LIN {X 0,Y 544.643,Z 479.184,A -85,B 0,C 180,E1 -3687.041,E2 -3687.041} C_VEL
LIN {X 0,Y 544.543,Z 480.909,A -85,B 0,C 180,E1 -3688.521,E2 -3688.521} C_VEL
LIN {X 0,Y 544.538,Z 481.5,A -85,B 0,C 180,E1 -3690,E2 -3690} C_VEL
LIN {X 0,Y 544.543,Z 480.907,A -85,B 0,C 180,E1 -3691.479,E2 -3691.479} C_VEL
LIN {X 0,Y 544.643,Z 479.179,A -85,B 0,C 180,E1 -3692.959,E2 -3692.959} C_VEL
LIN {X 0,Y 544.606,Z 476.288,A -85,B 0,C 180,E1 -3694.441,E2 -3694.441} C_VEL
LIN {X 0,Y 544.709,Z 472.165,A -85,B 0,C 180,E1 -3695.925,E2 -3695.925} C_VEL
LIN {X 0,Y 544.745,Z 466.7,A -85,B 0,C 180,E1 -3697.413,E2 -3697.413} C_VEL
LIN {X 0,Y 544.845,Z 459.743,A -85,B 0,C 180,E1 -3698.905,E2 -3698.905} C_VEL
LIN {X 0,Y 545.073,Z 451.08,A -85,B 0,C 180,E1 -3700.4,E2 -3700.4} C_VEL
LIN {X 0,Y 545.236,Z 441.69,A -85,B 0,C 180,E1 -3701.734,E2 -3701.734} C_VEL
LIN {X 0,Y 545.476,Z 432.34,A -85,B 0,C 180,E1 -3702.841,E2 -3702.841} C_VEL
LIN {X 0,Y 545.75,Z 421.005,A -85,B 0,C 180,E1 -3703.973,E2 -3703.973} C_VEL
LIN {X 0,Y 546.094,Z 408.349,A -85,B 0,C 180,E1 -3705.028,E2 -3705.028} C_VEL
LIN {X 0,Y 546.426,Z 394.866,A -85,B 0,C 180,E1 -3705.957,E2 -3705.957} C_VEL
LIN {X 0,Y 546.784,Z 381.388,A -85,B 0,C 180,E1 -3706.714,E2 -3706.714} C_VEL
LIN {X 0,Y 547.112,Z 366.588,A -85,B 0,C 180,E1 -3707.377,E2 -3707.377} C_VEL
LIN {X 0,Y 547.36,Z 351.136,A -85,B 0,C 180,E1 -3707.9,E2 -3707.9} C_VEL
LIN {X 0,Y 547.585,Z 335.478,A -85,B 0,C 180,E1 -3708.264,E2 -3708.264} C_VEL
LIN {X 0,Y 547.881,Z 279.91,A -85,B 0,C 180,E1 -3709.045,E2 -3709.045} C_VEL
LIN {X 0,Y 548.382,Z 177.465,A -85,B 0,C 180,E1 -3710.426,E2 -3710.426} C_VEL
LIN {X 0,Y 546.956,Z 166.898,A -85,B 0,C 180,E1 -3710.651,E2 -3710.651} C_VEL
LIN {X 0,Y 547.549,Z 134.253,A -85,B 0,C 180,E1 -3713.647,E2 -3713.647} C_VEL
LIN {X 0,Y 548.011,Z 115.051,A -85,B 0,C 180,E1 -3715.43,E2 -3715.43} C_VEL
LIN {X 0,Y 545.068,Z 103.217,A -85,B 0,C 180,E1 -3716.723,E2 -3716.723} C_VEL
LIN {X 0,Y 545.02,Z 103.223,A -85,B 0,C 180,E1 -3719.341,E2 -3719.341} C_VEL
LIN {X 0,Y 545.044,Z 103.214,A -85,B 0,C 180,E1 -3721.916,E2 -3721.916} C_VEL
LIN {X 0,Y 545.045,Z 103.216,A -85,B 0,C 180,E1 -3724.566,E2 -3724.566} C_VEL
LIN {X 0,Y 545.029,Z 103.22,A -85,B 0,C 180,E1 -3727.305,E2 -3727.305} C_VEL
LIN {X 0,Y 545.061,Z 103.212,A -85,B 0,C 180,E1 -3730.143,E2 -3730.143} C_VEL
LIN {X 0,Y 545.016,Z 103.22,A -85,B 0,C 180,E1 -3733.113,E2 -3733.113} C_VEL
LIN {X 0,Y 545.027,Z 103.216,A -85,B 0,C 180,E1 -3736.229,E2 -3736.229} C_VEL
LIN {X 0,Y 545.027,Z 103.22,A -85,B 0,C 180,E1 -3738.881,E2 -3738.881} C_VEL
LIN {X 0,Y 545.045,Z 103.214,A -85,B 0,C 180,E1 -3741.762,E2 -3741.762} C_VEL
LIN {X 0,Y 545.024,Z 103.223,A -85,B 0,C 180,E1 -3744.531,E2 -3744.531} C_VEL
LIN {X 0,Y 545.061,Z 103.212,A -85,B 0,C 180,E1 -3747.211,E2 -3747.211} C_VEL
LIN {X 0,Y 545.062,Z 103.213,A -85,B 0,C 180,E1 -3749.811,E2 -3749.811} C_VEL
LIN {X 0,Y 545.039,Z 103.217,A -85,B 0,C 180,E1 -3752.838,E2 -3752.838} C_VEL
LIN {X 0,Y 545.021,Z 103.22,A -85,B 0,C 180,E1 -3755.63,E2 -3755.63} C_VEL
LIN {X 0,Y 545.071,Z 103.293,A -85,B 0,C 180,E1 -3757.943,E2 -3757.943} C_VEL
LIN {X 0,Y 546.269,Z 110.508,A -85,B 0,C 180,E1 -3759.063,E2 -3759.063} C_VEL
LIN {X 0,Y 546.308,Z 113.04,A -85,B 0,C 180,E1 -3759.438,E2 -3759.438} C_VEL
LIN {X 0,Y 548.468,Z 123.652,A -85,B 0,C 180,E1 -3759.681,E2 -3759.681} C_VEL
LIN {X 0,Y 547.486,Z 277.991,A -85,B 0,C 180,E1 -3761.845,E2 -3761.845} C_VEL
LIN {X 0,Y 547.341,Z 292.858,A -85,B 0,C 180,E1 -3762.196,E2 -3762.196} C_VEL
LIN {X 0,Y 547.079,Z 308.282,A -85,B 0,C 180,E1 -3762.718,E2 -3762.718} C_VEL
LIN {X 0,Y 546.831,Z 321.071,A -85,B 0,C 180,E1 -3763.288,E2 -3763.288} C_VEL
LIN {X 0,Y 546.499,Z 334.745,A -85,B 0,C 180,E1 -3764.045,E2 -3764.045} C_VEL
LIN {X 0,Y 546.16,Z 348.31,A -85,B 0,C 180,E1 -3764.973,E2 -3764.973} C_VEL
LIN {X 0,Y 545.791,Z 360.976,A -85,B 0,C 180,E1 -3766.029,E2 -3766.029} C_VEL
LIN {X 0,Y 545.513,Z 372.228,A -85,B 0,C 180,E1 -3767.16,E2 -3767.16} C_VEL
LIN {X 0,Y 545.253,Z 382.568,A -85,B 0,C 180,E1 -3768.407,E2 -3768.407} C_VEL
LIN {X 0,Y 545.092,Z 390.911,A -85,B 0,C 180,E1 -3769.601,E2 -3769.601} C_VEL
LIN {X 0,Y 544.851,Z 399.516,A -85,B 0,C 180,E1 -3771.096,E2 -3771.096} C_VEL
LIN {X 0,Y 544.746,Z 406.525,A -85,B 0,C 180,E1 -3772.588,E2 -3772.588} C_VEL
LIN {X 0,Y 544.708,Z 411.986,A -85,B 0,C 180,E1 -3774.076,E2 -3774.076} C_VEL
LIN {X 0,Y 544.605,Z 416.188,A -85,B 0,C 180,E1 -3775.559,E2 -3775.559} C_VEL
LIN {X 0,Y 544.643,Z 419.108,A -85,B 0,C 180,E1 -3777.042,E2 -3777.042} C_VEL
LIN {X 0,Y 544.542,Z 420.838,A -85,B 0,C 180,E1 -3778.521,E2 -3778.521} C_VEL
LIN {X 0,Y 544.539,Z 421.496,A -85,B 0,C 180,E1 -3780,E2 -3780} C_VEL
LIN {X 0,Y 544.544,Z 420.915,A -85,B 0,C 180,E1 -3781.479,E2 -3781.479} C_VEL
LIN {X 0,Y 544.645,Z 419.238,A -85,B 0,C 180,E1 -3782.959,E2 -3782.959} C_VEL
LIN {X 0,Y 544.606,Z 416.423,A -85,B 0,C 180,E1 -3784.441,E2 -3784.441} C_VEL
LIN {X 0,Y 544.701,Z 412.267,A -85,B 0,C 180,E1 -3785.925,E2 -3785.925} C_VEL
LIN {X 0,Y 544.743,Z 406.901,A -85,B 0,C 180,E1 -3787.413,E2 -3787.413} C_VEL
LIN {X 0,Y 544.846,Z 399.966,A -85,B 0,C 180,E1 -3788.905,E2 -3788.905} C_VEL
LIN {X 0,Y 545.047,Z 392.645,A -85,B 0,C 180,E1 -3790.213,E2 -3790.213} C_VEL
LIN {X 0,Y 545.165,Z 383.552,A -85,B 0,C 180,E1 -3791.549,E2 -3791.549} C_VEL
LIN {X 0,Y 545.442,Z 374.644,A -85,B 0,C 180,E1 -3792.653,E2 -3792.653} C_VEL
LIN {X 0,Y 545.757,Z 362.903,A -85,B 0,C 180,E1 -3793.878,E2 -3793.878} C_VEL
LIN {X 0,Y 546.104,Z 350.94,A -85,B 0,C 180,E1 -3794.915,E2 -3794.915} C_VEL
LIN {X 0,Y 546.421,Z 337.749,A -85,B 0,C 180,E1 -3795.862,E2 -3795.862} C_VEL
LIN {X 0,Y 546.759,Z 324.87,A -85,B 0,C 180,E1 -3796.619,E2 -3796.619} C_VEL
LIN {X 0,Y 547.089,Z 310.858,A -85,B 0,C 180,E1 -3797.282,E2 -3797.282} C_VEL
LIN {X 0,Y 547.355,Z 295.027,A -85,B 0,C 180,E1 -3797.852,E2 -3797.852} C_VEL
LIN {X 0,Y 547.539,Z 279.859,A -85,B 0,C 180,E1 -3798.235,E2 -3798.235} C_VEL
LIN {X 0,Y 547.672,Z 258.394,A -85,B 0,C 180,E1 -3798.561,E2 -3798.561} C_VEL
LIN {X 0,Y 548.302,Z 149.592,A -85,B 0,C 180,E1 -3800.048,E2 -3800.048} C_VEL
LIN {X 0,Y 547.879,Z 143.779,A -85,B 0,C 180,E1 -3800.144,E2 -3800.144} C_VEL
LIN {X 0,Y 545.529,Z 134.425,A -85,B 0,C 180,E1 -3800.368,E2 -3800.368} C_VEL
LIN {X 0,Y 540.885,Z 119.579,A -85,B 0,C 180,E1 -3800.769,E2 -3800.769} C_VEL
LIN {X 0,Y 539.323,Z 112.564,A -85,B 0,C 180,E1 -3800.944,E2 -3800.944} C_VEL
LIN {X 0,Y 538.741,Z 107.608,A -85,B 0,C 180,E1 -3801.726,E2 -3801.726} C_VEL
LIN {X 0,Y 538.019,Z 104.095,A -85,B 0,C 180,E1 -3802.311,E2 -3802.311} C_VEL
LIN {X 0,Y 538.03,Z 104.093,A -85,B 0,C 180,E1 -3805.535,E2 -3805.535} C_VEL
LIN {X 0,Y 537.997,Z 104.095,A -85,B 0,C 180,E1 -3808.053,E2 -3808.053} C_VEL
LIN {X 0,Y 538.009,Z 104.089,A -85,B 0,C 180,E1 -3810.628,E2 -3810.628} C_VEL
LIN {X 0,Y 538.022,Z 104.092,A -85,B 0,C 180,E1 -3813.279,E2 -3813.279} C_VEL
LIN {X 0,Y 537.99,Z 104.094,A -85,B 0,C 180,E1 -3816.005,E2 -3816.005} C_VEL
LIN {X 0,Y 538.011,Z 104.089,A -85,B 0,C 180,E1 -3818.831,E2 -3818.831} C_VEL
LIN {X 0,Y 537.991,Z 104.093,A -85,B 0,C 180,E1 -3821.874,E2 -3821.874} C_VEL
LIN {X 0,Y 537.996,Z 104.091,A -85,B 0,C 180,E1 -3824.864,E2 -3824.864} C_VEL
LIN {X 0,Y 537.976,Z 104.093,A -85,B 0,C 180,E1 -3827.21,E2 -3827.21} C_VEL
LIN {X 0,Y 538.01,Z 104.088,A -85,B 0,C 180,E1 -3830.202,E2 -3830.202} C_VEL
LIN {X 0,Y 538.021,Z 104.092,A -85,B 0,C 180,E1 -3833.067,E2 -3833.067} C_VEL
LIN {X 0,Y 538,Z 104.088,A -85,B 0,C 180,E1 -3835.825,E2 -3835.825} C_VEL
LIN {X 0,Y 537.993,Z 104.093,A -85,B 0,C 180,E1 -3838.498,E2 -3838.498} C_VEL
LIN {X 0,Y 537.987,Z 104.096,A -85,B 0,C 180,E1 -3841.096,E2 -3841.096} C_VEL
LIN {X 0,Y 537.992,Z 104.091,A -85,B 0,C 180,E1 -3843.631,E2 -3843.631} C_VEL
LIN {X 0,Y 537.987,Z 104.089,A -85,B 0,C 180,E1 -3846.128,E2 -3846.128} C_VEL
LIN {X 0,Y 538.001,Z 104.097,A -85,B 0,C 180,E1 -3848.545,E2 -3848.545} C_VEL
LIN {X 0,Y 538.009,Z 104.094,A -85,B 0,C 180,E1 -3850.939,E2 -3850.939} C_VEL
LIN {X 0,Y 537.972,Z 104.092,A -85,B 0,C 180,E1 -3853.297,E2 -3853.297} C_VEL
LIN {X 0,Y 538.037,Z 104.086,A -85,B 0,C 180,E1 -3855.63,E2 -3855.63} C_VEL
LIN {X 0,Y 538.079,Z 104.084,A -85,B 0,C 180,E1 -3858.702,E2 -3858.702} C_VEL
LIN {X 0,Y 538.037,Z 104.087,A -85,B 0,C 180,E1 -3861.739,E2 -3861.739} C_VEL
LIN {X 0,Y 538.122,Z 104.079,A -85,B 0,C 180,E1 -3864.755,E2 -3864.755} C_VEL
LIN {X 0,Y 538.163,Z 104.075,A -85,B 0,C 180,E1 -3867.755,E2 -3867.755} C_VEL
LIN {X 0,Y 538.162,Z 104.078,A -85,B 0,C 180,E1 -3870,E2 -3870} C_VEL
LIN {X 0,Y 538.021,Z 104.191,A -85,B 0,C 180,E1 -3871.193,E2 -3871.193} C_VEL
LIN {X 0,Y 539.86,Z 112.82,A -85,B 0,C 180,E1 -3872.425,E2 -3872.425} C_VEL
LIN {X 0,Y 539.768,Z 126.914,A -85,B 0,C 180,E1 -3874.294,E2 -3874.294} C_VEL
LIN {X 0,Y 539.542,Z 141.011,A -85,B 0,C 180,E1 -3876.146,E2 -3876.146} C_VEL
LIN {X 0,Y 541.815,Z 152.663,A -85,B 0,C 180,E1 -3876.4,E2 -3876.4} C_VEL
LIN {X 0,Y 540.966,Z 306.907,A -85,B 0,C 180,E1 -3878.521,E2 -3878.521} C_VEL
LIN {X 0,Y 540.76,Z 321.623,A -85,B 0,C 180,E1 -3878.871,E2 -3878.871} C_VEL
LIN {X 0,Y 540.477,Z 336.09,A -85,B 0,C 180,E1 -3879.354,E2 -3879.354} C_VEL
LIN {X 0,Y 540.088,Z 351.048,A -85,B 0,C 180,E1 -3880.023,E2 -3880.023} C_VEL
LIN {X 0,Y 539.762,Z 362.973,A -85,B 0,C 180,E1 -3880.693,E2 -3880.693} C_VEL
LIN {X 0,Y 539.431,Z 374.357,A -85,B 0,C 180,E1 -3881.458,E2 -3881.458} C_VEL
LIN {X 0,Y 539.062,Z 385.999,A -85,B 0,C 180,E1 -3882.384,E2 -3882.384} C_VEL
LIN {X 0,Y 538.682,Z 398.586,A -85,B 0,C 180,E1 -3883.582,E2 -3883.582} C_VEL
LIN {X 0,Y 538.352,Z 407.929,A -85,B 0,C 180,E1 -3884.649,E2 -3884.649} C_VEL
LIN {X 0,Y 538.123,Z 416.015,A -85,B 0,C 180,E1 -3885.724,E2 -3885.724} C_VEL
LIN {X 0,Y 537.955,Z 423.592,A -85,B 0,C 180,E1 -3886.895,E2 -3886.895} C_VEL
LIN {X 0,Y 537.811,Z 430.113,A -85,B 0,C 180,E1 -3888.081,E2 -3888.081} C_VEL
LIN {X 0,Y 537.672,Z 436.272,A -85,B 0,C 180,E1 -3889.415,E2 -3889.415} C_VEL
LIN {X 0,Y 537.576,Z 442.31,A -85,B 0,C 180,E1 -3891.071,E2 -3891.071} C_VEL
LIN {X 0,Y 537.519,Z 445.693,A -85,B 0,C 180,E1 -3892.282,E2 -3892.282} C_VEL
LIN {X 0,Y 537.44,Z 448.666,A -85,B 0,C 180,E1 -3893.74,E2 -3893.74} C_VEL
LIN {X 0,Y 537.421,Z 450.12,A -85,B 0,C 180,E1 -3894.738,E2 -3894.738} C_VEL
LIN {X 0,Y 537.457,Z 450.902,A -85,B 0,C 180,E1 -3895.564,E2 -3895.564} C_VEL
LIN {X 0,Y 537.457,Z 451.454,A -85,B 0,C 180,E1 -3897.237,E2 -3897.237} C_VEL
LIN {X 0,Y 537.474,Z 450.617,A -85,B 0,C 180,E1 -3898.825,E2 -3898.825} C_VEL
LIN {X 0,Y 537.514,Z 448.664,A -85,B 0,C 180,E1 -3900.35,E2 -3900.35} C_VEL
LIN {X 0,Y 537.539,Z 445.699,A -85,B 0,C 180,E1 -3901.805,E2 -3901.805} C_VEL
LIN {X 0,Y 537.583,Z 441.423,A -85,B 0,C 180,E1 -3903.304,E2 -3903.304} C_VEL
LIN {X 0,Y 537.678,Z 435.709,A -85,B 0,C 180,E1 -3904.806,E2 -3904.806} C_VEL
LIN {X 0,Y 537.777,Z 430.06,A -85,B 0,C 180,E1 -3906.021,E2 -3906.021} C_VEL
LIN {X 0,Y 537.919,Z 423.829,A -85,B 0,C 180,E1 -3907.157,E2 -3907.157} C_VEL
LIN {X 0,Y 538.103,Z 417.58,A -85,B 0,C 180,E1 -3908.14,E2 -3908.14} C_VEL
LIN {X 0,Y 538.285,Z 409.15,A -85,B 0,C 180,E1 -3909.289,E2 -3909.289} C_VEL
LIN {X 0,Y 538.641,Z 398.911,A -85,B 0,C 180,E1 -3910.475,E2 -3910.475} C_VEL
LIN {X 0,Y 539.034,Z 386.361,A -85,B 0,C 180,E1 -3911.678,E2 -3911.678} C_VEL
LIN {X 0,Y 539.395,Z 375.415,A -85,B 0,C 180,E1 -3912.557,E2 -3912.557} C_VEL
LIN {X 0,Y 539.719,Z 364.092,A -85,B 0,C 180,E1 -3913.329,E2 -3913.329} C_VEL
LIN {X 0,Y 540.113,Z 350.528,A -85,B 0,C 180,E1 -3914.095,E2 -3914.095} C_VEL
LIN {X 0,Y 540.468,Z 336.169,A -85,B 0,C 180,E1 -3914.734,E2 -3914.734} C_VEL
LIN {X 0,Y 540.751,Z 321.821,A -85,B 0,C 180,E1 -3915.214,E2 -3915.214} C_VEL
LIN {X 0,Y 540.97,Z 308.257,A -85,B 0,C 180,E1 -3915.542,E2 -3915.542} C_VEL
LIN {X 0,Y 541.146,Z 275.268,A -85,B 0,C 180,E1 -3916.019,E2 -3916.019} C_VEL
LIN {X 0,Y 541.751,Z 148.68,A -85,B 0,C 180,E1 -3917.748,E2 -3917.748} C_VEL
LIN {X 0,Y 540.144,Z 139.429,A -85,B 0,C 180,E1 -3917.959,E2 -3917.959} C_VEL
LIN {X 0,Y 540.434,Z 114.155,A -85,B 0,C 180,E1 -3920.536,E2 -3920.536} C_VEL
LIN {X 0,Y 538.019,Z 104.094,A -85,B 0,C 180,E1 -3921.693,E2 -3921.693} C_VEL
LIN {X 0,Y 537.992,Z 104.098,A -85,B 0,C 180,E1 -3924.089,E2 -3924.089} C_VEL
LIN {X 0,Y 538.033,Z 104.088,A -85,B 0,C 180,E1 -3926.727,E2 -3926.727} C_VEL
LIN {X 0,Y 538.029,Z 104.093,A -85,B 0,C 180,E1 -3929.556,E2 -3929.556} C_VEL
LIN {X 0,Y 538.043,Z 104.09,A -85,B 0,C 180,E1 -3931.95,E2 -3931.95} C_VEL
LIN {X 0,Y 538.074,Z 104.083,A -85,B 0,C 180,E1 -3934.467,E2 -3934.467} C_VEL
LIN {X 0,Y 537.996,Z 104.099,A -85,B 0,C 180,E1 -3937.738,E2 -3937.738} C_VEL
LIN {X 0,Y 538.046,Z 104.233,A -85,B 0,C 180,E1 -3938.194,E2 -3938.194} C_VEL
LIN {X 0,Y 539.646,Z 111.177,A -85,B 0,C 180,E1 -3939.135,E2 -3939.135} C_VEL
LIN {X 0,Y 541.692,Z 120.025,A -85,B 0,C 180,E1 -3939.352,E2 -3939.352} C_VEL
LIN {X 0,Y 541.213,Z 211.695,A -85,B 0,C 180,E1 -3940.662,E2 -3940.662} C_VEL
LIN {X 0,Y 540.755,Z 277.646,A -85,B 0,C 180,E1 -3941.593,E2 -3941.593} C_VEL
LIN {X 0,Y 540.575,Z 293.955,A -85,B 0,C 180,E1 -3941.99,E2 -3941.99} C_VEL
LIN {X 0,Y 540.278,Z 308.349,A -85,B 0,C 180,E1 -3942.493,E2 -3942.493} C_VEL
LIN {X 0,Y 540.006,Z 321.097,A -85,B 0,C 180,E1 -3943.07,E2 -3943.07} C_VEL
LIN {X 0,Y 539.638,Z 334.778,A -85,B 0,C 180,E1 -3943.836,E2 -3943.836} C_VEL
LIN {X 0,Y 539.285,Z 348.853,A -85,B 0,C 180,E1 -3944.815,E2 -3944.815} C_VEL
LIN {X 0,Y 538.903,Z 359.967,A -85,B 0,C 180,E1 -3945.75,E2 -3945.75} C_VEL
LIN {X 0,Y 538.607,Z 370.522,A -85,B 0,C 180,E1 -3946.8,E2 -3946.8} C_VEL
LIN {X 0,Y 538.31,Z 380.347,A -85,B 0,C 180,E1 -3947.942,E2 -3947.942} C_VEL
LIN {X 0,Y 538.072,Z 391.099,A -85,B 0,C 180,E1 -3949.463,E2 -3949.463} C_VEL
LIN {X 0,Y 537.856,Z 397.775,A -85,B 0,C 180,E1 -3950.599,E2 -3950.599} C_VEL
LIN {X 0,Y 537.768,Z 403.459,A -85,B 0,C 180,E1 -3951.734,E2 -3951.734} C_VEL
LIN {X 0,Y 537.679,Z 408.25,A -85,B 0,C 180,E1 -3952.867,E2 -3952.867} C_VEL
LIN {X 0,Y 537.643,Z 413.347,A -85,B 0,C 180,E1 -3954.373,E2 -3954.373} C_VEL
LIN {X 0,Y 537.562,Z 418,A -85,B 0,C 180,E1 -3956.252,E2 -3956.252} C_VEL
LIN {X 0,Y 537.488,Z 420.262,A -85,B 0,C 180,E1 -3957.752,E2 -3957.752} C_VEL
LIN {X 0,Y 537.439,Z 421.392,A -85,B 0,C 180,E1 -3959.25,E2 -3959.25} C_VEL
LIN {X 0,Y 537.441,Z 421.625,A -85,B 0,C 180,E1 -3960,E2 -3960} C_VEL
LIN {X 0,Y 537.449,Z 421.076,A -85,B 0,C 180,E1 -3961.498,E2 -3961.498} C_VEL
LIN {X 0,Y 537.574,Z 419.381,A -85,B 0,C 180,E1 -3962.997,E2 -3962.997} C_VEL
LIN {X 0,Y 537.562,Z 418.182,A -85,B 0,C 180,E1 -3963.748,E2 -3963.748} C_VEL
LIN {X 0,Y 537.643,Z 413.645,A -85,B 0,C 180,E1 -3965.626,E2 -3965.626} C_VEL
LIN {X 0,Y 537.68,Z 408.627,A -85,B 0,C 180,E1 -3967.133,E2 -3967.133} C_VEL
LIN {X 0,Y 537.778,Z 402.213,A -85,B 0,C 180,E1 -3968.643,E2 -3968.643} C_VEL
LIN {X 0,Y 537.984,Z 394.053,A -85,B 0,C 180,E1 -3970.157,E2 -3970.157} C_VEL
LIN {X 0,Y 538.09,Z 386.69,A -85,B 0,C 180,E1 -3971.298,E2 -3971.298} C_VEL
LIN {X 0,Y 538.374,Z 378.069,A -85,B 0,C 180,E1 -3972.438,E2 -3972.438} C_VEL
LIN {X 0,Y 538.7,Z 367.876,A -85,B 0,C 180,E1 -3973.582,E2 -3973.582} C_VEL
LIN {X 0,Y 539.029,Z 355.64,A -85,B 0,C 180,E1 -3974.729,E2 -3974.729} C_VEL
LIN {X 0,Y 539.411,Z 343.304,A -85,B 0,C 180,E1 -3975.683,E2 -3975.683} C_VEL
LIN {X 0,Y 539.757,Z 329.755,A -85,B 0,C 180,E1 -3976.548,E2 -3976.548} C_VEL
LIN {X 0,Y 540.09,Z 315.713,A -85,B 0,C 180,E1 -3977.268,E2 -3977.268} C_VEL
LIN {X 0,Y 540.388,Z 300.471,A -85,B 0,C 180,E1 -3977.869,E2 -3977.869} C_VEL
LIN {X 0,Y 540.641,Z 284.928,A -85,B 0,C 180,E1 -3978.312,E2 -3978.312} C_VEL
LIN {X 0,Y 540.764,Z 268.903,A -85,B 0,C 180,E1 -3978.602,E2 -3978.602} C_VEL
LIN {X 0,Y 541.688,Z 140.378,A -85,B 0,C 180,E1 -3980.429,E2 -3980.429} C_VEL
LIN {X 0,Y 541.716,Z 123.174,A -85,B 0,C 180,E1 -3980.691,E2 -3980.691} C_VEL
LIN {X 0,Y 539.622,Z 114.321,A -85,B 0,C 180,E1 -3980.928,E2 -3980.928} C_VEL
LIN {X 0,Y 539.443,Z 110.534,A -85,B 0,C 180,E1 -3981.567,E2 -3981.567} C_VEL
LIN {X 0,Y 537.987,Z 104.098,A -85,B 0,C 180,E1 -3982.768,E2 -3982.768} C_VEL
LIN {X 0,Y 538.007,Z 104.097,A -85,B 0,C 180,E1 -3985.664,E2 -3985.664} C_VEL
LIN {X 0,Y 537.996,Z 104.097,A -85,B 0,C 180,E1 -3988.052,E2 -3988.052} C_VEL
LIN {X 0,Y 538.007,Z 104.091,A -85,B 0,C 180,E1 -3990.628,E2 -3990.628} C_VEL
LIN {X 0,Y 538.019,Z 104.094,A -85,B 0,C 180,E1 -3993.278,E2 -3993.278} C_VEL
LIN {X 0,Y 537.987,Z 104.095,A -85,B 0,C 180,E1 -3996.005,E2 -3996.005} C_VEL
LIN {X 0,Y 538.008,Z 104.092,A -85,B 0,C 180,E1 -3998.831,E2 -3998.831} C_VEL
LIN {X 0,Y 537.987,Z 104.095,A -85,B 0,C 180,E1 -4001.873,E2 -4001.873} C_VEL
LIN {X 0,Y 537.993,Z 104.096,A -85,B 0,C 180,E1 -4004.863,E2 -4004.863} C_VEL
LIN {X 0,Y 537.973,Z 104.101,A -85,B 0,C 180,E1 -4007.209,E2 -4007.209} C_VEL
LIN {X 0,Y 538.006,Z 104.091,A -85,B 0,C 180,E1 -4010.201,E2 -4010.201} C_VEL
LIN {X 0,Y 538.016,Z 104.097,A -85,B 0,C 180,E1 -4013.066,E2 -4013.066} C_VEL
LIN {X 0,Y 537.995,Z 104.093,A -85,B 0,C 180,E1 -4015.825,E2 -4015.825} C_VEL
LIN {X 0,Y 537.988,Z 104.099,A -85,B 0,C 180,E1 -4018.497,E2 -4018.497} C_VEL
LIN {X 0,Y 537.984,Z 104.119,A -85,B 0,C 180,E1 -4021.415,E2 -4021.415} C_VEL
LIN {X 0,Y 540.297,Z 114.01,A -85,B 0,C 180,E1 -4022.774,E2 -4022.774} C_VEL
LIN {X 0,Y 540.209,Z 127.243,A -85,B 0,C 180,E1 -4024.389,E2 -4024.389} C_VEL
LIN {X 0,Y 539.701,Z 152.43,A -85,B 0,C 180,E1 -4027.372,E2 -4027.372} C_VEL
LIN {X 0,Y 539.403,Z 167.004,A -85,B 0,C 180,E1 -4029.066,E2 -4029.066} C_VEL
LIN {X 0,Y 541.666,Z 181.231,A -85,B 0,C 180,E1 -4029.388,E2 -4029.388} C_VEL
LIN {X 0,Y 540.901,Z 297.15,A -85,B 0,C 180,E1 -4031.02,E2 -4031.02} C_VEL
LIN {X 0,Y 540.627,Z 336.129,A -85,B 0,C 180,E1 -4031.586,E2 -4031.586} C_VEL
LIN {X 0,Y 540.429,Z 351.514,A -85,B 0,C 180,E1 -4031.961,E2 -4031.961} C_VEL
LIN {X 0,Y 540.147,Z 365.617,A -85,B 0,C 180,E1 -4032.44,E2 -4032.44} C_VEL
LIN {X 0,Y 539.837,Z 379.671,A -85,B 0,C 180,E1 -4033.065,E2 -4033.065} C_VEL
LIN {X 0,Y 539.411,Z 393.424,A -85,B 0,C 180,E1 -4033.83,E2 -4033.83} C_VEL
LIN {X 0,Y 539.106,Z 407.383,A -85,B 0,C 180,E1 -4034.787,E2 -4034.787} C_VEL
LIN {X 0,Y 538.733,Z 420.06,A -85,B 0,C 180,E1 -4035.842,E2 -4035.842} C_VEL
LIN {X 0,Y 538.433,Z 431.551,A -85,B 0,C 180,E1 -4036.988,E2 -4036.988} C_VEL
LIN {X 0,Y 538.148,Z 442.074,A -85,B 0,C 180,E1 -4038.241,E2 -4038.241} C_VEL
LIN {X 0,Y 537.985,Z 451.91,A -85,B 0,C 180,E1 -4039.652,E2 -4039.652} C_VEL
LIN {X 0,Y 537.797,Z 459.537,A -85,B 0,C 180,E1 -4040.978,E2 -4040.978} C_VEL
LIN {X 0,Y 537.661,Z 466.643,A -85,B 0,C 180,E1 -4042.489,E2 -4042.489} C_VEL
LIN {X 0,Y 537.623,Z 472.161,A -85,B 0,C 180,E1 -4043.997,E2 -4043.997} C_VEL
LIN {X 0,Y 537.508,Z 476.29,A -85,B 0,C 180,E1 -4045.5,E2 -4045.5} C_VEL
LIN {X 0,Y 537.543,Z 479.183,A -85,B 0,C 180,E1 -4047.002,E2 -4047.002} C_VEL
LIN {X 0,Y 537.448,Z 480.909,A -85,B 0,C 180,E1 -4048.501,E2 -4048.501} C_VEL
LIN {X 0,Y 537.439,Z 481.5,A -85,B 0,C 180,E1 -4050,E2 -4050} C_VEL
LIN {X 0,Y 537.448,Z 480.906,A -85,B 0,C 180,E1 -4051.499,E2 -4051.499} C_VEL
LIN {X 0,Y 537.543,Z 479.178,A -85,B 0,C 180,E1 -4052.998,E2 -4052.998} C_VEL
LIN {X 0,Y 537.508,Z 476.287,A -85,B 0,C 180,E1 -4054.5,E2 -4054.5} C_VEL
LIN {X 0,Y 537.623,Z 472.165,A -85,B 0,C 180,E1 -4056.003,E2 -4056.003} C_VEL
LIN {X 0,Y 537.661,Z 466.645,A -85,B 0,C 180,E1 -4057.511,E2 -4057.511} C_VEL
LIN {X 0,Y 537.797,Z 459.558,A -85,B 0,C 180,E1 -4059.022,E2 -4059.022} C_VEL
LIN {X 0,Y 538.005,Z 450.726,A -85,B 0,C 180,E1 -4060.538,E2 -4060.538} C_VEL
LIN {X 0,Y 538.204,Z 440.976,A -85,B 0,C 180,E1 -4061.912,E2 -4061.912} C_VEL
LIN {X 0,Y 538.443,Z 431.755,A -85,B 0,C 180,E1 -4063.012,E2 -4063.012} C_VEL
LIN {X 0,Y 538.75,Z 420.377,A -85,B 0,C 180,E1 -4064.158,E2 -4064.158} C_VEL
LIN {X 0,Y 539.138,Z 407.558,A -85,B 0,C 180,E1 -4065.234,E2 -4065.234} C_VEL
LIN {X 0,Y 539.487,Z 394.091,A -85,B 0,C 180,E1 -4066.168,E2 -4066.168} C_VEL
LIN {X 0,Y 539.877,Z 380.546,A -85,B 0,C 180,E1 -4066.934,E2 -4066.934} C_VEL
LIN {X 0,Y 540.246,Z 365.604,A -85,B 0,C 180,E1 -4067.605,E2 -4067.605} C_VEL
LIN {X 0,Y 540.543,Z 349.885,A -85,B 0,C 180,E1 -4068.133,E2 -4068.133} C_VEL
LIN {X 0,Y 540.789,Z 334.296,A -85,B 0,C 180,E1 -4068.492,E2 -4068.492} C_VEL
LIN {X 0,Y 541.185,Z 271.432,A -85,B 0,C 180,E1 -4069.388,E2 -4069.388} C_VEL
LIN {X 0,Y 541.704,Z 178.455,A -85,B 0,C 180,E1 -4070.669,E2 -4070.669} C_VEL
LIN {X 0,Y 540.108,Z 166.532,A -85,B 0,C 180,E1 -4070.93,E2 -4070.93} C_VEL
LIN {X 0,Y 540.802,Z 134.049,A -85,B 0,C 180,E1 -4073.952,E2 -4073.952} C_VEL
LIN {X 0,Y 541.258,Z 117.243,A -85,B 0,C 180,E1 -4075.531,E2 -4075.531} C_VEL
LIN {X 0,Y 539.353,Z 109.176,A -85,B 0,C 180,E1 -4076.402,E2 -4076.402} C_VEL
LIN {X 0,Y 538.011,Z 104.097,A -85,B 0,C 180,E1 -4076.97,E2 -4076.97} C_VEL
LIN {X 0,Y 537.996,Z 104.094,A -85,B 0,C 180,E1 -4079.762,E2 -4079.762} C_VEL
LIN {X 0,Y 538.01,Z 104.091,A -85,B 0,C 180,E1 -4082.383,E2 -4082.383} C_VEL
LIN {X 0,Y 537.985,Z 104.099,A -85,B 0,C 180,E1 -4085.085,E2 -4085.085} C_VEL
LIN {X 0,Y 537.986,Z 104.093,A -85,B 0,C 180,E1 -4087.878,E2 -4087.878} C_VEL
LIN {X 0,Y 538.001,Z 104.097,A -85,B 0,C 180,E1 -4090.78,E2 -4090.78} C_VEL
LIN {X 0,Y 538,Z 104.09,A -85,B 0,C 180,E1 -4094.071,E2 -4094.071} C_VEL
LIN {X 0,Y 537.97,Z 104.098,A -85,B 0,C 180,E1 -4097.019,E2 -4097.019} C_VEL
LIN {X 0,Y 538.005,Z 104.091,A -85,B 0,C 180,E1 -4099.258,E2 -4099.258} C_VEL
LIN {X 0,Y 537.986,Z 104.096,A -85,B 0,C 180,E1 -4102.122,E2 -4102.122} C_VEL
LIN {X 0,Y 537.986,Z 104.096,A -85,B 0,C 180,E1 -4104.915,E2 -4104.915} C_VEL
LIN {X 0,Y 538.014,Z 104.09,A -85,B 0,C 180,E1 -4107.617,E2 -4107.617} C_VEL
LIN {X 0,Y 537.999,Z 104.098,A -85,B 0,C 180,E1 -4110.238,E2 -4110.238} C_VEL
LIN {X 0,Y 538.012,Z 104.094,A -85,B 0,C 180,E1 -4112.793,E2 -4112.793} C_VEL
LIN {X 0,Y 537.983,Z 104.096,A -85,B 0,C 180,E1 -4115.29,E2 -4115.29} C_VEL
LIN {X 0,Y 538.049,Z 104.182,A -85,B 0,C 180,E1 -4117.741,E2 -4117.741} C_VEL
LIN {X 0,Y 539.422,Z 111.104,A -85,B 0,C 180,E1 -4118.805,E2 -4118.805} C_VEL
LIN {X 0,Y 539.539,Z 113.837,A -85,B 0,C 180,E1 -4119.183,E2 -4119.183} C_VEL
LIN {X 0,Y 541.81,Z 124.5,A -85,B 0,C 180,E1 -4119.436,E2 -4119.436} C_VEL
LIN {X 0,Y 540.676,Z 277.84,A -85,B 0,C 180,E1 -4121.636,E2 -4121.636} C_VEL
LIN {X 0,Y 540.517,Z 293.642,A -85,B 0,C 180,E1 -4122.013,E2 -4122.013} C_VEL
LIN {X 0,Y 540.223,Z 307.729,A -85,B 0,C 180,E1 -4122.492,E2 -4122.492} C_VEL
LIN {X 0,Y 539.988,Z 320.75,A -85,B 0,C 180,E1 -4123.07,E2 -4123.07} C_VEL
LIN {X 0,Y 539.636,Z 334.584,A -85,B 0,C 180,E1 -4123.837,E2 -4123.837} C_VEL
LIN {X 0,Y 539.231,Z 348.235,A -85,B 0,C 180,E1 -4124.773,E2 -4124.773} C_VEL
LIN {X 0,Y 538.87,Z 361.028,A -85,B 0,C 180,E1 -4125.846,E2 -4125.846} C_VEL
LIN {X 0,Y 538.563,Z 372.359,A -85,B 0,C 180,E1 -4126.991,E2 -4126.991} C_VEL
LIN {X 0,Y 538.288,Z 381.878,A -85,B 0,C 180,E1 -4128.134,E2 -4128.134} C_VEL
LIN {X 0,Y 538.075,Z 391.161,A -85,B 0,C 180,E1 -4129.464,E2 -4129.464} C_VEL
LIN {X 0,Y 537.81,Z 399.848,A -85,B 0,C 180,E1 -4130.978,E2 -4130.978} C_VEL
LIN {X 0,Y 537.695,Z 406.816,A -85,B 0,C 180,E1 -4132.49,E2 -4132.49} C_VEL
LIN {X 0,Y 537.644,Z 412.255,A -85,B 0,C 180,E1 -4133.998,E2 -4133.998} C_VEL
LIN {X 0,Y 537.514,Z 416.402,A -85,B 0,C 180,E1 -4135.501,E2 -4135.501} C_VEL
LIN {X 0,Y 537.572,Z 419.272,A -85,B 0,C 180,E1 -4137.003,E2 -4137.003} C_VEL
LIN {X 0,Y 537.448,Z 420.979,A -85,B 0,C 180,E1 -4138.502,E2 -4138.502} C_VEL
LIN {X 0,Y 537.441,Z 421.618,A -85,B 0,C 180,E1 -4140,E2 -4140} C_VEL
LIN {X 0,Y 537.449,Z 421.048,A -85,B 0,C 180,E1 -4141.499,E2 -4141.499} C_VEL
LIN {X 0,Y 537.574,Z 419.388,A -85,B 0,C 180,E1 -4142.998,E2 -4142.998} C_VEL
LIN {X 0,Y 537.513,Z 416.595,A -85,B 0,C 180,E1 -4144.5,E2 -4144.5} C_VEL
LIN {X 0,Y 537.618,Z 412.497,A -85,B 0,C 180,E1 -4146.003,E2 -4146.003} C_VEL
LIN {X 0,Y 537.674,Z 407.15,A -85,B 0,C 180,E1 -4147.511,E2 -4147.511} C_VEL
LIN {X 0,Y 537.797,Z 400.241,A -85,B 0,C 180,E1 -4149.022,E2 -4149.022} C_VEL
LIN {X 0,Y 538.02,Z 392.87,A -85,B 0,C 180,E1 -4150.347,E2 -4150.347} C_VEL
LIN {X 0,Y 538.206,Z 383.355,A -85,B 0,C 180,E1 -4151.753,E2 -4151.753} C_VEL
LIN {X 0,Y 538.527,Z 373.119,A -85,B 0,C 180,E1 -4153.01,E2 -4153.01} C_VEL
LIN {X 0,Y 538.848,Z 361.97,A -85,B 0,C 180,E1 -4154.155,E2 -4154.155} C_VEL
LIN {X 0,Y 539.217,Z 349.459,A -85,B 0,C 180,E1 -4155.226,E2 -4155.226} C_VEL
LIN {X 0,Y 539.613,Z 336.15,A -85,B 0,C 180,E1 -4156.164,E2 -4156.164} C_VEL
LIN {X 0,Y 539.968,Z 322.83,A -85,B 0,C 180,E1 -4156.932,E2 -4156.932} C_VEL
LIN {X 0,Y 540.286,Z 309.339,A -85,B 0,C 180,E1 -4157.555,E2 -4157.555} C_VEL
LIN {X 0,Y 540.558,Z 294.398,A -85,B 0,C 180,E1 -4158.084,E2 -4158.084} C_VEL
LIN {X 0,Y 540.764,Z 278.839,A -85,B 0,C 180,E1 -4158.47,E2 -4158.47} C_VEL
LIN {X 0,Y 540.936,Z 250.852,A -85,B 0,C 180,E1 -4158.884,E2 -4158.884} C_VEL
LIN {X 0,Y 541.813,Z 124.079,A -85,B 0,C 180,E1 -4160.665,E2 -4160.665} C_VEL
LIN {X 0,Y 540.885,Z 119.579,A -85,B 0,C 180,E1 -4160.769,E2 -4160.769} C_VEL
LIN {X 0,Y 539.445,Z 116.158,A -85,B 0,C 180,E1 -4160.917,E2 -4160.917} C_VEL
LIN {X 0,Y 537.33,Z 113.451,A -85,B 0,C 180,E1 -4161.145,E2 -4161.145} C_VEL
LIN {X 0,Y 534.298,Z 110.59,A -85,B 0,C 180,E1 -4161.534,E2 -4161.534} C_VEL
LIN {X 0,Y 531.889,Z 107.931,A -85,B 0,C 180,E1 -4161.994,E2 -4161.994} C_VEL
LIN {X 0,Y 531.277,Z 106.472,A -85,B 0,C 180,E1 -4162.24,E2 -4162.24} C_VEL
LIN {X 0,Y 530.988,Z 104.97,A -85,B 0,C 180,E1 -4162.51,E2 -4162.51} C_VEL
LIN {X 0,Y 530.97,Z 104.974,A -85,B 0,C 180,E1 -4165.834,E2 -4165.834} C_VEL
LIN {X 0,Y 530.959,Z 104.968,A -85,B 0,C 180,E1 -4168.458,E2 -4168.458} C_VEL
LIN {X 0,Y 530.953,Z 104.97,A -85,B 0,C 180,E1 -4171.08,E2 -4171.08} C_VEL
LIN {X 0,Y 530.952,Z 104.974,A -85,B 0,C 180,E1 -4173.776,E2 -4173.776} C_VEL
LIN {X 0,Y 530.952,Z 104.968,A -85,B 0,C 180,E1 -4176.559,E2 -4176.559} C_VEL
LIN {X 0,Y 530.972,Z 104.974,A -85,B 0,C 180,E1 -4179.445,E2 -4179.445} C_VEL
LIN {X 0,Y 530.92,Z 104.972,A -85,B 0,C 180,E1 -4182.463,E2 -4182.463} C_VEL
LIN {X 0,Y 530.966,Z 104.965,A -85,B 0,C 180,E1 -4185.451,E2 -4185.451} C_VEL
LIN {X 0,Y 530.961,Z 104.964,A -85,B 0,C 180,E1 -4188.561,E2 -4188.561} C_VEL
LIN {X 0,Y 530.954,Z 104.97,A -85,B 0,C 180,E1 -4191.529,E2 -4191.529} C_VEL
LIN {X 0,Y 530.949,Z 104.962,A -85,B 0,C 180,E1 -4194.379,E2 -4194.379} C_VEL
LIN {X 0,Y 530.967,Z 104.973,A -85,B 0,C 180,E1 -4197.133,E2 -4197.133} C_VEL
LIN {X 0,Y 530.937,Z 104.966,A -85,B 0,C 180,E1 -4199.801,E2 -4199.801} C_VEL
LIN {X 0,Y 530.965,Z 104.968,A -85,B 0,C 180,E1 -4202.478,E2 -4202.478} C_VEL
LIN {X 0,Y 530.95,Z 104.971,A -85,B 0,C 180,E1 -4204.94,E2 -4204.94} C_VEL
LIN {X 0,Y 530.954,Z 104.97,A -85,B 0,C 180,E1 -4208.246,E2 -4208.246} C_VEL
LIN {X 0,Y 530.965,Z 104.972,A -85,B 0,C 180,E1 -4210.676,E2 -4210.676} C_VEL
LIN {X 0,Y 530.94,Z 104.97,A -85,B 0,C 180,E1 -4213.069,E2 -4213.069} C_VEL
LIN {X 0,Y 530.999,Z 104.963,A -85,B 0,C 180,E1 -4215.435,E2 -4215.435} C_VEL
LIN {X 0,Y 531.038,Z 104.964,A -85,B 0,C 180,E1 -4218.55,E2 -4218.55} C_VEL
LIN {X 0,Y 530.986,Z 104.965,A -85,B 0,C 180,E1 -4221.628,E2 -4221.628} C_VEL
LIN {X 0,Y 531.083,Z 104.957,A -85,B 0,C 180,E1 -4224.685,E2 -4224.685} C_VEL
LIN {X 0,Y 531.135,Z 104.951,A -85,B 0,C 180,E1 -4227.725,E2 -4227.725} C_VEL
LIN {X 0,Y 531.13,Z 104.953,A -85,B 0,C 180,E1 -4230,E2 -4230} C_VEL
LIN {X 0,Y 530.965,Z 105.073,A -85,B 0,C 180,E1 -4230.972,E2 -4230.972} C_VEL
LIN {X 0,Y 532.948,Z 114.075,A -85,B 0,C 180,E1 -4232.267,E2 -4232.267} C_VEL
LIN {X 0,Y 533.051,Z 121.105,A -85,B 0,C 180,E1 -4233.212,E2 -4233.212} C_VEL
LIN {X 0,Y 532.691,Z 141.284,A -85,B 0,C 180,E1 -4235.869,E2 -4235.869} C_VEL
LIN {X 0,Y 535.084,Z 152.452,A -85,B 0,C 180,E1 -4236.126,E2 -4236.126} C_VEL
LIN {X 0,Y 534.245,Z 306.512,A -85,B 0,C 180,E1 -4238.273,E2 -4238.273} C_VEL
LIN {X 0,Y 534.018,Z 321.293,A -85,B 0,C 180,E1 -4238.622,E2 -4238.622} C_VEL
LIN {X 0,Y 533.717,Z 335.348,A -85,B 0,C 180,E1 -4239.092,E2 -4239.092} C_VEL
LIN {X 0,Y 533.321,Z 350.547,A -85,B 0,C 180,E1 -4239.768,E2 -4239.768} C_VEL
LIN {X 0,Y 532.885,Z 364.156,A -85,B 0,C 180,E1 -4240.544,E2 -4240.544} C_VEL
LIN {X 0,Y 532.533,Z 375.433,A -85,B 0,C 180,E1 -4241.321,E2 -4241.321} C_VEL
LIN {X 0,Y 532.134,Z 386.503,A -85,B 0,C 180,E1 -4242.221,E2 -4242.221} C_VEL
LIN {X 0,Y 531.738,Z 398.462,A -85,B 0,C 180,E1 -4243.374,E2 -4243.374} C_VEL
LIN {X 0,Y 531.35,Z 408.651,A -85,B 0,C 180,E1 -4244.555,E2 -4244.555} C_VEL
LIN {X 0,Y 531.082,Z 417.324,A -85,B 0,C 180,E1 -4245.741,E2 -4245.741} C_VEL
LIN {X 0,Y 530.915,Z 424.777,A -85,B 0,C 180,E1 -4246.931,E2 -4246.931} C_VEL
LIN {X 0,Y 530.681,Z 433.098,A -85,B 0,C 180,E1 -4248.532,E2 -4248.532} C_VEL
LIN {X 0,Y 530.583,Z 438.647,A -85,B 0,C 180,E1 -4249.871,E2 -4249.871} C_VEL
LIN {X 0,Y 530.489,Z 443.575,A -85,B 0,C 180,E1 -4251.366,E2 -4251.366} C_VEL
LIN {X 0,Y 530.422,Z 446.717,A -85,B 0,C 180,E1 -4252.597,E2 -4252.597} C_VEL
LIN {X 0,Y 530.356,Z 449.155,A -85,B 0,C 180,E1 -4253.885,E2 -4253.885} C_VEL
LIN {X 0,Y 530.362,Z 451.229,A -85,B 0,C 180,E1 -4255.697,E2 -4255.697} C_VEL
LIN {X 0,Y 530.37,Z 451.592,A -85,B 0,C 180,E1 -4257.398,E2 -4257.398} C_VEL
LIN {X 0,Y 530.386,Z 450.663,A -85,B 0,C 180,E1 -4259.008,E2 -4259.008} C_VEL
LIN {X 0,Y 530.431,Z 448.625,A -85,B 0,C 180,E1 -4260.545,E2 -4260.545} C_VEL
LIN {X 0,Y 530.466,Z 445.565,A -85,B 0,C 180,E1 -4262.013,E2 -4262.013} C_VEL
LIN {X 0,Y 530.539,Z 440.13,A -85,B 0,C 180,E1 -4263.805,E2 -4263.805} C_VEL
LIN {X 0,Y 530.658,Z 434.722,A -85,B 0,C 180,E1 -4265.186,E2 -4265.186} C_VEL
LIN {X 0,Y 530.818,Z 426.97,A -85,B 0,C 180,E1 -4266.781,E2 -4266.781} C_VEL
LIN {X 0,Y 531.078,Z 418.23,A -85,B 0,C 180,E1 -4268.219,E2 -4268.219} C_VEL
LIN {X 0,Y 531.293,Z 409.611,A -85,B 0,C 180,E1 -4269.416,E2 -4269.416} C_VEL
LIN {X 0,Y 531.674,Z 399.402,A -85,B 0,C 180,E1 -4270.618,E2 -4270.618} C_VEL
LIN {X 0,Y 532.118,Z 386.943,A -85,B 0,C 180,E1 -4271.835,E2 -4271.835} C_VEL
LIN {X 0,Y 532.492,Z 376.505,A -85,B 0,C 180,E1 -4272.693,E2 -4272.693} C_VEL
LIN {X 0,Y 532.905,Z 363.891,A -85,B 0,C 180,E1 -4273.565,E2 -4273.565} C_VEL
LIN {X 0,Y 533.358,Z 349.739,A -85,B 0,C 180,E1 -4274.366,E2 -4274.366} C_VEL
LIN {X 0,Y 533.712,Z 334.66,A -85,B 0,C 180,E1 -4275.026,E2 -4275.026} C_VEL
LIN {X 0,Y 534.041,Z 319.893,A -85,B 0,C 180,E1 -4275.509,E2 -4275.509} C_VEL
LIN {X 0,Y 534.234,Z 304.541,A -85,B 0,C 180,E1 -4275.853,E2 -4275.853} C_VEL
LIN {X 0,Y 535.221,Z 150.298,A -85,B 0,C 180,E1 -4277.988,E2 -4277.988} C_VEL
LIN {X 0,Y 533.316,Z 139.395,A -85,B 0,C 180,E1 -4278.244,E2 -4278.244} C_VEL
LIN {X 0,Y 533.71,Z 116.918,A -85,B 0,C 180,E1 -4280.556,E2 -4280.556} C_VEL
LIN {X 0,Y 531.67,Z 107.843,A -85,B 0,C 180,E1 -4281.59,E2 -4281.59} C_VEL
LIN {X 0,Y 530.97,Z 104.972,A -85,B 0,C 180,E1 -4281.953,E2 -4281.953} C_VEL
LIN {X 0,Y 530.971,Z 104.968,A -85,B 0,C 180,E1 -4285.149,E2 -4285.149} C_VEL
LIN {X 0,Y 530.97,Z 104.972,A -85,B 0,C 180,E1 -4288.032,E2 -4288.032} C_VEL
LIN {X 0,Y 530.992,Z 104.963,A -85,B 0,C 180,E1 -4290.874,E2 -4290.874} C_VEL
LIN {X 0,Y 531.005,Z 104.968,A -85,B 0,C 180,E1 -4293.256,E2 -4293.256} C_VEL
LIN {X 0,Y 530.987,Z 104.968,A -85,B 0,C 180,E1 -4295.961,E2 -4295.961} C_VEL
LIN {X 0,Y 530.993,Z 104.983,A -85,B 0,C 180,E1 -4297.951,E2 -4297.951} C_VEL
LIN {X 0,Y 532.511,Z 111.461,A -85,B 0,C 180,E1 -4298.838,E2 -4298.838} C_VEL
LIN {X 0,Y 534.24,Z 117.068,A -85,B 0,C 180,E1 -4299.003,E2 -4299.003} C_VEL
LIN {X 0,Y 535.183,Z 123.212,A -85,B 0,C 180,E1 -4299.136,E2 -4299.136} C_VEL
LIN {X 0,Y 533.983,Z 277.963,A -85,B 0,C 180,E1 -4301.375,E2 -4301.375} C_VEL
LIN {X 0,Y 533.78,Z 294.25,A -85,B 0,C 180,E1 -4301.777,E2 -4301.777} C_VEL
LIN {X 0,Y 533.451,Z 309.259,A -85,B 0,C 180,E1 -4302.311,E2 -4302.311} C_VEL
LIN {X 0,Y 533.143,Z 322.862,A -85,B 0,C 180,E1 -4302.944,E2 -4302.944} C_VEL
LIN {X 0,Y 532.738,Z 336.273,A -85,B 0,C 180,E1 -4303.72,E2 -4303.72} C_VEL
LIN {X 0,Y 532.35,Z 349.833,A -85,B 0,C 180,E1 -4304.69,E2 -4304.69} C_VEL
LIN {X 0,Y 531.956,Z 361.092,A -85,B 0,C 180,E1 -4305.657,E2 -4305.657} C_VEL
LIN {X 0,Y 531.658,Z 370.653,A -85,B 0,C 180,E1 -4306.624,E2 -4306.624} C_VEL
LIN {X 0,Y 531.326,Z 380.517,A -85,B 0,C 180,E1 -4307.781,E2 -4307.781} C_VEL
LIN {X 0,Y 531.085,Z 390.112,A -85,B 0,C 180,E1 -4309.13,E2 -4309.13} C_VEL
LIN {X 0,Y 530.825,Z 398.041,A -85,B 0,C 180,E1 -4310.474,E2 -4310.474} C_VEL
LIN {X 0,Y 530.732,Z 403.764,A -85,B 0,C 180,E1 -4311.624,E2 -4311.624} C_VEL
LIN {X 0,Y 530.618,Z 408.572,A -85,B 0,C 180,E1 -4312.771,E2 -4312.771} C_VEL
LIN {X 0,Y 530.571,Z 413.7,A -85,B 0,C 180,E1 -4314.298,E2 -4314.298} C_VEL
LIN {X 0,Y 530.433,Z 416.702,A -85,B 0,C 180,E1 -4315.44,E2 -4315.44} C_VEL
LIN {X 0,Y 530.481,Z 418.355,A -85,B 0,C 180,E1 -4316.202,E2 -4316.202} C_VEL
LIN {X 0,Y 530.41,Z 420.66,A -85,B 0,C 180,E1 -4317.722,E2 -4317.722} C_VEL
LIN {X 0,Y 530.351,Z 421.803,A -85,B 0,C 180,E1 -4319.24,E2 -4319.24} C_VEL
LIN {X 0,Y 530.353,Z 422.023,A -85,B 0,C 180,E1 -4320,E2 -4320} C_VEL
LIN {X 0,Y 530.363,Z 421.492,A -85,B 0,C 180,E1 -4321.518,E2 -4321.518} C_VEL
LIN {X 0,Y 530.505,Z 419.794,A -85,B 0,C 180,E1 -4323.037,E2 -4323.037} C_VEL
LIN {X 0,Y 530.449,Z 416.96,A -85,B 0,C 180,E1 -4324.559,E2 -4324.559} C_VEL
LIN {X 0,Y 530.596,Z 412.927,A -85,B 0,C 180,E1 -4326.082,E2 -4326.082} C_VEL
LIN {X 0,Y 530.63,Z 407.555,A -85,B 0,C 180,E1 -4327.611,E2 -4327.611} C_VEL
LIN {X 0,Y 530.756,Z 400.623,A -85,B 0,C 180,E1 -4329.143,E2 -4329.143} C_VEL
LIN {X 0,Y 530.999,Z 393.193,A -85,B 0,C 180,E1 -4330.485,E2 -4330.485} C_VEL
LIN {X 0,Y 531.234,Z 383.848,A -85,B 0,C 180,E1 -4331.889,E2 -4331.889} C_VEL
LIN {X 0,Y 531.591,Z 373.381,A -85,B 0,C 180,E1 -4333.182,E2 -4333.182} C_VEL
LIN {X 0,Y 531.92,Z 362.138,A -85,B 0,C 180,E1 -4334.343,E2 -4334.343} C_VEL
LIN {X 0,Y 532.357,Z 349.848,A -85,B 0,C 180,E1 -4335.401,E2 -4335.401} C_VEL
LIN {X 0,Y 532.696,Z 337.518,A -85,B 0,C 180,E1 -4336.281,E2 -4336.281} C_VEL
LIN {X 0,Y 533.089,Z 324.236,A -85,B 0,C 180,E1 -4337.057,E2 -4337.057} C_VEL
LIN {X 0,Y 533.38,Z 310.741,A -85,B 0,C 180,E1 -4337.691,E2 -4337.691} C_VEL
LIN {X 0,Y 533.657,Z 295.888,A -85,B 0,C 180,E1 -4338.226,E2 -4338.226} C_VEL
LIN {X 0,Y 533.827,Z 281.495,A -85,B 0,C 180,E1 -4338.598,E2 -4338.598} C_VEL
LIN {X 0,Y 533.944,Z 260.301,A -85,B 0,C 180,E1 -4338.937,E2 -4338.937} C_VEL
LIN {X 0,Y 535.003,Z 143.872,A -85,B 0,C 180,E1 -4340.637,E2 -4340.637} C_VEL
LIN {X 0,Y 535.034,Z 124.294,A -85,B 0,C 180,E1 -4340.941,E2 -4340.941} C_VEL
LIN {X 0,Y 532.798,Z 114.968,A -85,B 0,C 180,E1 -4341.201,E2 -4341.201} C_VEL
LIN {X 0,Y 532.594,Z 112.165,A -85,B 0,C 180,E1 -4341.683,E2 -4341.683} C_VEL
LIN {X 0,Y 530.986,Z 104.971,A -85,B 0,C 180,E1 -4343.034,E2 -4343.034} C_VEL
LIN {X 0,Y 530.971,Z 104.974,A -85,B 0,C 180,E1 -4345.899,E2 -4345.899} C_VEL
LIN {X 0,Y 530.957,Z 104.971,A -85,B 0,C 180,E1 -4348.458,E2 -4348.458} C_VEL
LIN {X 0,Y 530.951,Z 104.972,A -85,B 0,C 180,E1 -4351.079,E2 -4351.079} C_VEL
LIN {X 0,Y 530.95,Z 104.975,A -85,B 0,C 180,E1 -4353.775,E2 -4353.775} C_VEL
LIN {X 0,Y 530.949,Z 104.97,A -85,B 0,C 180,E1 -4356.559,E2 -4356.559} C_VEL
LIN {X 0,Y 530.982,Z 104.972,A -85,B 0,C 180,E1 -4359.444,E2 -4359.444} C_VEL
LIN {X 0,Y 530.917,Z 104.974,A -85,B 0,C 180,E1 -4362.463,E2 -4362.463} C_VEL
LIN {X 0,Y 530.962,Z 104.973,A -85,B 0,C 180,E1 -4365.45,E2 -4365.45} C_VEL
LIN {X 0,Y 530.957,Z 104.97,A -85,B 0,C 180,E1 -4368.561,E2 -4368.561} C_VEL
LIN {X 0,Y 530.95,Z 104.972,A -85,B 0,C 180,E1 -4371.529,E2 -4371.529} C_VEL
LIN {X 0,Y 530.933,Z 104.975,A -85,B 0,C 180,E1 -4374.378,E2 -4374.378} C_VEL
LIN {X 0,Y 530.963,Z 104.974,A -85,B 0,C 180,E1 -4377.133,E2 -4377.133} C_VEL
LIN {X 0,Y 530.928,Z 104.978,A -85,B 0,C 180,E1 -4379.8,E2 -4379.8} C_VEL
LIN {X 0,Y 530.954,Z 104.997,A -85,B 0,C 180,E1 -4381.138,E2 -4381.138} C_VEL
LIN {X 0,Y 533.58,Z 116.565,A -85,B 0,C 180,E1 -4382.761,E2 -4382.761} C_VEL
LIN {X 0,Y 533.168,Z 137.334,A -85,B 0,C 180,E1 -4385.316,E2 -4385.316} C_VEL
LIN {X 0,Y 532.535,Z 162.459,A -85,B 0,C 180,E1 -4388.314,E2 -4388.314} C_VEL
LIN {X 0,Y 532.458,Z 166.478,A -85,B 0,C 180,E1 -4388.787,E2 -4388.787} C_VEL
LIN {X 0,Y 534.992,Z 181.708,A -85,B 0,C 180,E1 -4389.135,E2 -4389.135} C_VEL
LIN {X 0,Y 534.07,Z 297.737,A -85,B 0,C 180,E1 -4390.818,E2 -4390.818} C_VEL
LIN {X 0,Y 533.791,Z 335.667,A -85,B 0,C 180,E1 -4391.381,E2 -4391.381} C_VEL
LIN {X 0,Y 533.561,Z 350.566,A -85,B 0,C 180,E1 -4391.745,E2 -4391.745} C_VEL
LIN {X 0,Y 533.255,Z 365.364,A -85,B 0,C 180,E1 -4392.255,E2 -4392.255} C_VEL
LIN {X 0,Y 532.906,Z 378.372,A -85,B 0,C 180,E1 -4392.837,E2 -4392.837} C_VEL
LIN {X 0,Y 532.499,Z 392.31,A -85,B 0,C 180,E1 -4393.614,E2 -4393.614} C_VEL
LIN {X 0,Y 532.186,Z 405.126,A -85,B 0,C 180,E1 -4394.49,E2 -4394.49} C_VEL
LIN {X 0,Y 531.796,Z 416.988,A -85,B 0,C 180,E1 -4395.458,E2 -4395.458} C_VEL
LIN {X 0,Y 531.518,Z 427.11,A -85,B 0,C 180,E1 -4396.426,E2 -4396.426} C_VEL
LIN {X 0,Y 531.199,Z 437.437,A -85,B 0,C 180,E1 -4397.585,E2 -4397.585} C_VEL
LIN {X 0,Y 530.989,Z 447.499,A -85,B 0,C 180,E1 -4398.935,E2 -4398.935} C_VEL
LIN {X 0,Y 530.745,Z 455.864,A -85,B 0,C 180,E1 -4400.28,E2 -4400.28} C_VEL
LIN {X 0,Y 530.65,Z 462.748,A -85,B 0,C 180,E1 -4401.623,E2 -4401.623} C_VEL
LIN {X 0,Y 530.549,Z 469.105,A -85,B 0,C 180,E1 -4403.153,E2 -4403.153} C_VEL
LIN {X 0,Y 530.509,Z 474.015,A -85,B 0,C 180,E1 -4404.679,E2 -4404.679} C_VEL
LIN {X 0,Y 530.481,Z 477.605,A -85,B 0,C 180,E1 -4406.202,E2 -4406.202} C_VEL
LIN {X 0,Y 530.409,Z 479.959,A -85,B 0,C 180,E1 -4407.722,E2 -4407.722} C_VEL
LIN {X 0,Y 530.341,Z 481.142,A -85,B 0,C 180,E1 -4409.241,E2 -4409.241} C_VEL
LIN {X 0,Y 530.341,Z 481.143,A -85,B 0,C 180,E1 -4410.759,E2 -4410.759} C_VEL
LIN {X 0,Y 530.409,Z 479.964,A -85,B 0,C 180,E1 -4412.278,E2 -4412.278} C_VEL
LIN {X 0,Y 530.481,Z 477.62,A -85,B 0,C 180,E1 -4413.798,E2 -4413.798} C_VEL
LIN {X 0,Y 530.509,Z 474.053,A -85,B 0,C 180,E1 -4415.321,E2 -4415.321} C_VEL
LIN {X 0,Y 530.569,Z 469.174,A -85,B 0,C 180,E1 -4416.847,E2 -4416.847} C_VEL
LIN {X 0,Y 530.664,Z 462.845,A -85,B 0,C 180,E1 -4418.377,E2 -4418.377} C_VEL
LIN {X 0,Y 530.804,Z 454.885,A -85,B 0,C 180,E1 -4419.911,E2 -4419.911} C_VEL
LIN {X 0,Y 531,Z 446.402,A -85,B 0,C 180,E1 -4421.258,E2 -4421.258} C_VEL
LIN {X 0,Y 531.26,Z 436.166,A -85,B 0,C 180,E1 -4422.608,E2 -4422.608} C_VEL
LIN {X 0,Y 531.579,Z 425.709,A -85,B 0,C 180,E1 -4423.767,E2 -4423.767} C_VEL
LIN {X 0,Y 531.989,Z 413.175,A -85,B 0,C 180,E1 -4424.928,E2 -4424.928} C_VEL
LIN {X 0,Y 532.376,Z 400.615,A -85,B 0,C 180,E1 -4425.898,E2 -4425.898} C_VEL
LIN {X 0,Y 532.812,Z 386.863,A -85,B 0,C 180,E1 -4426.771,E2 -4426.771} C_VEL
LIN {X 0,Y 533.181,Z 372.63,A -85,B 0,C 180,E1 -4427.5,E2 -4427.5} C_VEL
LIN {X 0,Y 533.591,Z 358.027,A -85,B 0,C 180,E1 -4428.08,E2 -4428.08} C_VEL
LIN {X 0,Y 533.838,Z 342.585,A -85,B 0,C 180,E1 -4428.531,E2 -4428.531} C_VEL
LIN {X 0,Y 533.99,Z 327.026,A -85,B 0,C 180,E1 -4428.826,E2 -4428.826} C_VEL
LIN {X 0,Y 534.581,Z 246.742,A -85,B 0,C 180,E1 -4429.963,E2 -4429.963} C_VEL
LIN {X 0,Y 535.041,Z 181.129,A -85,B 0,C 180,E1 -4430.893,E2 -4430.893} C_VEL
LIN {X 0,Y 534.679,Z 175.935,A -85,B 0,C 180,E1 -4430.988,E2 -4430.988} C_VEL
LIN {X 0,Y 533.271,Z 166.251,A -85,B 0,C 180,E1 -4431.209,E2 -4431.209} C_VEL
LIN {X 0,Y 533.988,Z 135.801,A -85,B 0,C 180,E1 -4434.079,E2 -4434.079} C_VEL
LIN {X 0,Y 534.492,Z 118.622,A -85,B 0,C 180,E1 -4435.716,E2 -4435.716} C_VEL
LIN {X 0,Y 530.982,Z 104.973,A -85,B 0,C 180,E1 -4437.258,E2 -4437.258} C_VEL
LIN {X 0,Y 530.945,Z 104.971,A -85,B 0,C 180,E1 -4440.199,E2 -4440.199} C_VEL
LIN {X 0,Y 530.964,Z 104.973,A -85,B 0,C 180,E1 -4442.867,E2 -4442.867} C_VEL
LIN {X 0,Y 530.945,Z 104.971,A -85,B 0,C 180,E1 -4445.621,E2 -4445.621} C_VEL
LIN {X 0,Y 530.961,Z 104.973,A -85,B 0,C 180,E1 -4448.653,E2 -4448.653} C_VEL
LIN {X 0,Y 530.957,Z 104.969,A -85,B 0,C 180,E1 -4451.439,E2 -4451.439} C_VEL
LIN {X 0,Y 530.962,Z 104.971,A -85,B 0,C 180,E1 -4454.55,E2 -4454.55} C_VEL
LIN {X 0,Y 530.917,Z 104.972,A -85,B 0,C 180,E1 -4457.537,E2 -4457.537} C_VEL
LIN {X 0,Y 530.968,Z 104.973,A -85,B 0,C 180,E1 -4460.555,E2 -4460.555} C_VEL
LIN {X 0,Y 530.949,Z 104.97,A -85,B 0,C 180,E1 -4463.441,E2 -4463.441} C_VEL
LIN {X 0,Y 530.96,Z 104.975,A -85,B 0,C 180,E1 -4466.501,E2 -4466.501} C_VEL
LIN {X 0,Y 530.961,Z 104.969,A -85,B 0,C 180,E1 -4469.358,E2 -4469.358} C_VEL
LIN {X 0,Y 530.964,Z 104.974,A -85,B 0,C 180,E1 -4472.478,E2 -4472.478} C_VEL
LIN {X 0,Y 530.95,Z 104.973,A -85,B 0,C 180,E1 -4474.94,E2 -4474.94} C_VEL
LIN {X 0,Y 531.012,Z 105.119,A -85,B 0,C 180,E1 -4477.523,E2 -4477.523} C_VEL
LIN {X 0,Y 532.616,Z 113.895,A -85,B 0,C 180,E1 -4478.881,E2 -4478.881} C_VEL
LIN {X 0,Y 535.144,Z 125.261,A -85,B 0,C 180,E1 -4479.182,E2 -4479.182} C_VEL
LIN {X 0,Y 534.024,Z 251.83,A -85,B 0,C 180,E1 -4481.038,E2 -4481.038} C_VEL
LIN {X 0,Y 533.87,Z 279.895,A -85,B 0,C 180,E1 -4481.464,E2 -4481.464} C_VEL
LIN {X 0,Y 533.648,Z 295.248,A -85,B 0,C 180,E1 -4481.848,E2 -4481.848} C_VEL
LIN {X 0,Y 533.353,Z 310.883,A -85,B 0,C 180,E1 -4482.408,E2 -4482.408} C_VEL
LIN {X 0,Y 533.051,Z 324.263,A -85,B 0,C 180,E1 -4483.04,E2 -4483.04} C_VEL
LIN {X 0,Y 532.672,Z 337.506,A -85,B 0,C 180,E1 -4483.816,E2 -4483.816} C_VEL
LIN {X 0,Y 532.27,Z 350.996,A -85,B 0,C 180,E1 -4484.786,E2 -4484.786} C_VEL
LIN {X 0,Y 531.882,Z 363.179,A -85,B 0,C 180,E1 -4485.851,E2 -4485.851} C_VEL
LIN {X 0,Y 531.526,Z 374.24,A -85,B 0,C 180,E1 -4487.01,E2 -4487.01} C_VEL
LIN {X 0,Y 531.223,Z 384.071,A -85,B 0,C 180,E1 -4488.24,E2 -4488.24} C_VEL
LIN {X 0,Y 531.016,Z 392.609,A -85,B 0,C 180,E1 -4489.515,E2 -4489.515} C_VEL
LIN {X 0,Y 530.769,Z 400.136,A -85,B 0,C 180,E1 -4490.858,E2 -4490.858} C_VEL
LIN {X 0,Y 530.632,Z 407.133,A -85,B 0,C 180,E1 -4492.389,E2 -4492.389} C_VEL
LIN {X 0,Y 530.588,Z 412.618,A -85,B 0,C 180,E1 -4493.917,E2 -4493.917} C_VEL
LIN {X 0,Y 530.434,Z 416.765,A -85,B 0,C 180,E1 -4495.441,E2 -4495.441} C_VEL
LIN {X 0,Y 530.503,Z 419.654,A -85,B 0,C 180,E1 -4496.963,E2 -4496.963} C_VEL
LIN {X 0,Y 530.362,Z 421.394,A -85,B 0,C 180,E1 -4498.482,E2 -4498.482} C_VEL
LIN {X 0,Y 530.352,Z 422.003,A -85,B 0,C 180,E1 -4500,E2 -4500} C_VEL
LIN {X 0,Y 530.362,Z 421.449,A -85,B 0,C 180,E1 -4501.519,E2 -4501.519} C_VEL
LIN {X 0,Y 530.505,Z 419.756,A -85,B 0,C 180,E1 -4503.038,E2 -4503.038} C_VEL
LIN {X 0,Y 530.43,Z 416.922,A -85,B 0,C 180,E1 -4504.56,E2 -4504.56} C_VEL
LIN {X 0,Y 530.564,Z 412.833,A -85,B 0,C 180,E1 -4506.083,E2 -4506.083} C_VEL
LIN {X 0,Y 530.613,Z 407.418,A -85,B 0,C 180,E1 -4507.611,E2 -4507.611} C_VEL
LIN {X 0,Y 530.756,Z 400.5,A -85,B 0,C 180,E1 -4509.143,E2 -4509.143} C_VEL
LIN {X 0,Y 531.003,Z 393.064,A -85,B 0,C 180,E1 -4510.486,E2 -4510.486} C_VEL
LIN {X 0,Y 531.142,Z 384.945,A -85,B 0,C 180,E1 -4511.718,E2 -4511.718} C_VEL
LIN {X 0,Y 531.514,Z 374.923,A -85,B 0,C 180,E1 -4512.99,E2 -4512.99} C_VEL
LIN {X 0,Y 531.889,Z 363.049,A -85,B 0,C 180,E1 -4514.247,E2 -4514.247} C_VEL
LIN {X 0,Y 532.285,Z 350.924,A -85,B 0,C 180,E1 -4515.312,E2 -4515.312} C_VEL
LIN {X 0,Y 532.714,Z 337.558,A -85,B 0,C 180,E1 -4516.281,E2 -4516.281} C_VEL
LIN {X 0,Y 533.072,Z 324.502,A -85,B 0,C 180,E1 -4517.058,E2 -4517.058} C_VEL
LIN {X 0,Y 533.449,Z 310.174,A -85,B 0,C 180,E1 -4517.738,E2 -4517.738} C_VEL
LIN {X 0,Y 533.75,Z 295.446,A -85,B 0,C 180,E1 -4518.273,E2 -4518.273} C_VEL
LIN {X 0,Y 533.982,Z 280.415,A -85,B 0,C 180,E1 -4518.662,E2 -4518.662} C_VEL
LIN {X 0,Y 534.121,Z 258.421,A -85,B 0,C 180,E1 -4519.006,E2 -4519.006} C_VEL
LIN {X 0,Y 535.121,Z 124.653,A -85,B 0,C 180,E1 -4520.927,E2 -4520.927} C_VEL
LIN {X 0,Y 532.438,Z 112.87,A -85,B 0,C 180,E1 -4521.221,E2 -4521.221} C_VEL
LIN {X 0,Y 531.277,Z 106.472,A -85,B 0,C 180,E1 -4522.24,E2 -4522.24} C_VEL
LIN {X 0,Y 530.677,Z 105.358,A -85,B 0,C 180,E1 -4522.561,E2 -4522.561} C_VEL
LIN {X 0,Y 529.537,Z 105.149,A -85,B 0,C 180,E1 -4523.004,E2 -4523.004} C_VEL
LIN {X 0,Y 524.883,Z 105.865,A -85,B 0,C 180,E1 -4524.685,E2 -4524.685} C_VEL
LIN {X 0,Y 523.975,Z 105.858,A -85,B 0,C 180,E1 -4525.35,E2 -4525.35} C_VEL
LIN {X 0,Y 523.906,Z 105.851,A -85,B 0,C 180,E1 -4525.574,E2 -4525.574} C_VEL
LIN {X 0,Y 523.912,Z 105.851,A -85,B 0,C 180,E1 -4528.003,E2 -4528.003} C_VEL
LIN {X 0,Y 523.937,Z 105.843,A -85,B 0,C 180,E1 -4530.853,E2 -4530.853} C_VEL
LIN {X 0,Y 523.928,Z 105.85,A -85,B 0,C 180,E1 -4533.729,E2 -4533.729} C_VEL
LIN {X 0,Y 523.9,Z 105.846,A -85,B 0,C 180,E1 -4536.401,E2 -4536.401} C_VEL
LIN {X 0,Y 523.914,Z 105.848,A -85,B 0,C 180,E1 -4539.086,E2 -4539.086} C_VEL
LIN {X 0,Y 523.901,Z 105.847,A -85,B 0,C 180,E1 -4542.124,E2 -4542.124} C_VEL
LIN {X 0,Y 523.936,Z 105.842,A -85,B 0,C 180,E1 -4545.311,E2 -4545.311} C_VEL
LIN {X 0,Y 523.922,Z 105.842,A -85,B 0,C 180,E1 -4548.695,E2 -4548.695} C_VEL
LIN {X 0,Y 523.914,Z 105.844,A -85,B 0,C 180,E1 -4551.898,E2 -4551.898} C_VEL
LIN {X 0,Y 523.92,Z 105.843,A -85,B 0,C 180,E1 -4554.913,E2 -4554.913} C_VEL
LIN {X 0,Y 523.933,Z 105.843,A -85,B 0,C 180,E1 -4557.681,E2 -4557.681} C_VEL
LIN {X 0,Y 523.934,Z 105.844,A -85,B 0,C 180,E1 -4560.681,E2 -4560.681} C_VEL
LIN {X 0,Y 523.905,Z 105.846,A -85,B 0,C 180,E1 -4563.725,E2 -4563.725} C_VEL
LIN {X 0,Y 523.9,Z 105.844,A -85,B 0,C 180,E1 -4566.269,E2 -4566.269} C_VEL
LIN {X 0,Y 523.926,Z 105.849,A -85,B 0,C 180,E1 -4568.766,E2 -4568.766} C_VEL
LIN {X 0,Y 523.929,Z 105.845,A -85,B 0,C 180,E1 -4571.22,E2 -4571.22} C_VEL
LIN {X 0,Y 523.883,Z 105.847,A -85,B 0,C 180,E1 -4573.637,E2 -4573.637} C_VEL
LIN {X 0,Y 523.963,Z 105.84,A -85,B 0,C 180,E1 -4575.235,E2 -4575.235} C_VEL
LIN {X 0,Y 524.018,Z 105.84,A -85,B 0,C 180,E1 -4578.394,E2 -4578.394} C_VEL
LIN {X 0,Y 523.949,Z 105.841,A -85,B 0,C 180,E1 -4581.515,E2 -4581.515} C_VEL
LIN {X 0,Y 524.03,Z 105.836,A -85,B 0,C 180,E1 -4584.613,E2 -4584.613} C_VEL
LIN {X 0,Y 524.105,Z 105.826,A -85,B 0,C 180,E1 -4587.694,E2 -4587.694} C_VEL
LIN {X 0,Y 523.977,Z 105.844,A -85,B 0,C 180,E1 -4590.384,E2 -4590.384} C_VEL
LIN {X 0,Y 523.91,Z 105.957,A -85,B 0,C 180,E1 -4590.745,E2 -4590.745} C_VEL
LIN {X 0,Y 526.236,Z 116.667,A -85,B 0,C 180,E1 -4592.296,E2 -4592.296} C_VEL
LIN {X 0,Y 525.902,Z 136.749,A -85,B 0,C 180,E1 -4594.983,E2 -4594.983} C_VEL
LIN {X 0,Y 525.779,Z 141.103,A -85,B 0,C 180,E1 -4595.561,E2 -4595.561} C_VEL
LIN {X 0,Y 528.467,Z 153.532,A -85,B 0,C 180,E1 -4595.868,E2 -4595.868} C_VEL
LIN {X 0,Y 527.507,Z 307.359,A -85,B 0,C 180,E1 -4598.042,E2 -4598.042} C_VEL
LIN {X 0,Y 527.283,Z 322.315,A -85,B 0,C 180,E1 -4598.407,E2 -4598.407} C_VEL
LIN {X 0,Y 526.906,Z 337.698,A -85,B 0,C 180,E1 -4598.944,E2 -4598.944} C_VEL
LIN {X 0,Y 526.492,Z 351.892,A -85,B 0,C 180,E1 -4599.605,E2 -4599.605} C_VEL
LIN {X 0,Y 526.021,Z 365.331,A -85,B 0,C 180,E1 -4600.391,E2 -4600.391} C_VEL
LIN {X 0,Y 525.549,Z 377.815,A -85,B 0,C 180,E1 -4601.278,E2 -4601.278} C_VEL
LIN {X 0,Y 525.053,Z 391.441,A -85,B 0,C 180,E1 -4602.465,E2 -4602.465} C_VEL
LIN {X 0,Y 524.65,Z 401.885,A -85,B 0,C 180,E1 -4603.558,E2 -4603.558} C_VEL
LIN {X 0,Y 524.295,Z 411.649,A -85,B 0,C 180,E1 -4604.755,E2 -4604.755} C_VEL
LIN {X 0,Y 523.953,Z 421.232,A -85,B 0,C 180,E1 -4606.16,E2 -4606.16} C_VEL
LIN {X 0,Y 523.758,Z 428.394,A -85,B 0,C 180,E1 -4607.422,E2 -4607.422} C_VEL
LIN {X 0,Y 523.607,Z 434.885,A -85,B 0,C 180,E1 -4608.792,E2 -4608.792} C_VEL
LIN {X 0,Y 523.504,Z 439.589,A -85,B 0,C 180,E1 -4609.99,E2 -4609.99} C_VEL
LIN {X 0,Y 523.4,Z 443.674,A -85,B 0,C 180,E1 -4611.257,E2 -4611.257} C_VEL
LIN {X 0,Y 523.372,Z 445.934,A -85,B 0,C 180,E1 -4612.095,E2 -4612.095} C_VEL
LIN {X 0,Y 523.268,Z 449.224,A -85,B 0,C 180,E1 -4613.761,E2 -4613.761} C_VEL
LIN {X 0,Y 523.238,Z 450.43,A -85,B 0,C 180,E1 -4614.607,E2 -4614.607} C_VEL
LIN {X 0,Y 523.248,Z 451.673,A -85,B 0,C 180,E1 -4616.311,E2 -4616.311} C_VEL
LIN {X 0,Y 523.269,Z 451.738,A -85,B 0,C 180,E1 -4617.57,E2 -4617.57} C_VEL
LIN {X 0,Y 523.313,Z 450.709,A -85,B 0,C 180,E1 -4619.197,E2 -4619.197} C_VEL
LIN {X 0,Y 523.347,Z 448.578,A -85,B 0,C 180,E1 -4620.744,E2 -4620.744} C_VEL
LIN {X 0,Y 523.4,Z 444.668,A -85,B 0,C 180,E1 -4622.487,E2 -4622.487} C_VEL
LIN {X 0,Y 523.467,Z 440.118,A -85,B 0,C 180,E1 -4623.955,E2 -4623.955} C_VEL
LIN {X 0,Y 523.611,Z 434.113,A -85,B 0,C 180,E1 -4625.486,E2 -4625.486} C_VEL
LIN {X 0,Y 523.828,Z 425.893,A -85,B 0,C 180,E1 -4627.139,E2 -4627.139} C_VEL
LIN {X 0,Y 524.05,Z 418.645,A -85,B 0,C 180,E1 -4628.335,E2 -4628.335} C_VEL
LIN {X 0,Y 524.303,Z 410.071,A -85,B 0,C 180,E1 -4629.547,E2 -4629.547} C_VEL
LIN {X 0,Y 524.735,Z 399.684,A -85,B 0,C 180,E1 -4630.789,E2 -4630.789} C_VEL
LIN {X 0,Y 525.211,Z 387.527,A -85,B 0,C 180,E1 -4631.995,E2 -4631.995} C_VEL
LIN {X 0,Y 525.643,Z 375.492,A -85,B 0,C 180,E1 -4632.991,E2 -4632.991} C_VEL
LIN {X 0,Y 526.166,Z 362.121,A -85,B 0,C 180,E1 -4633.907,E2 -4633.907} C_VEL
LIN {X 0,Y 526.617,Z 348.102,A -85,B 0,C 180,E1 -4634.68,E2 -4634.68} C_VEL
LIN {X 0,Y 526.967,Z 334.728,A -85,B 0,C 180,E1 -4635.265,E2 -4635.265} C_VEL
LIN {X 0,Y 527.319,Z 319.502,A -85,B 0,C 180,E1 -4635.766,E2 -4635.766} C_VEL
LIN {X 0,Y 527.53,Z 304.607,A -85,B 0,C 180,E1 -4636.098,E2 -4636.098} C_VEL
LIN {X 0,Y 528.602,Z 151.204,A -85,B 0,C 180,E1 -4638.249,E2 -4638.249} C_VEL
LIN {X 0,Y 526.508,Z 139.441,A -85,B 0,C 180,E1 -4638.526,E2 -4638.526} C_VEL
LIN {X 0,Y 526.861,Z 118.16,A -85,B 0,C 180,E1 -4640.74,E2 -4640.74} C_VEL
LIN {X 0,Y 523.942,Z 105.85,A -85,B 0,C 180,E1 -4642.187,E2 -4642.187} C_VEL
LIN {X 0,Y 523.926,Z 105.846,A -85,B 0,C 180,E1 -4644.911,E2 -4644.911} C_VEL
LIN {X 0,Y 523.938,Z 105.849,A -85,B 0,C 180,E1 -4647.679,E2 -4647.679} C_VEL
LIN {X 0,Y 523.957,Z 105.839,A -85,B 0,C 180,E1 -4650.676,E2 -4650.676} C_VEL
LIN {X 0,Y 523.977,Z 105.843,A -85,B 0,C 180,E1 -4653.728,E2 -4653.728} C_VEL
LIN {X 0,Y 523.928,Z 105.847,A -85,B 0,C 180,E1 -4656.27,E2 -4656.27} C_VEL
LIN {X 0,Y 523.97,Z 106.047,A -85,B 0,C 180,E1 -4657.743,E2 -4657.743} C_VEL
LIN {X 0,Y 525.44,Z 112.095,A -85,B 0,C 180,E1 -4658.554,E2 -4658.554} C_VEL
LIN {X 0,Y 527.803,Z 119.025,A -85,B 0,C 180,E1 -4658.763,E2 -4658.763} C_VEL
LIN {X 0,Y 528.545,Z 123.003,A -85,B 0,C 180,E1 -4658.857,E2 -4658.857} C_VEL
LIN {X 0,Y 527.389,Z 256.47,A -85,B 0,C 180,E1 -4660.818,E2 -4660.818} C_VEL
LIN {X 0,Y 527.213,Z 280.51,A -85,B 0,C 180,E1 -4661.2,E2 -4661.2} C_VEL
LIN {X 0,Y 526.965,Z 296.062,A -85,B 0,C 180,E1 -4661.609,E2 -4661.609} C_VEL
LIN {X 0,Y 526.623,Z 310.137,A -85,B 0,C 180,E1 -4662.125,E2 -4662.125} C_VEL
LIN {X 0,Y 526.256,Z 324.528,A -85,B 0,C 180,E1 -4662.814,E2 -4662.814} C_VEL
LIN {X 0,Y 525.826,Z 337.681,A -85,B 0,C 180,E1 -4663.599,E2 -4663.599} C_VEL
LIN {X 0,Y 525.421,Z 351.061,A -85,B 0,C 180,E1 -4664.582,E2 -4664.582} C_VEL
LIN {X 0,Y 524.938,Z 363.24,A -85,B 0,C 180,E1 -4665.659,E2 -4665.659} C_VEL
LIN {X 0,Y 524.575,Z 374.319,A -85,B 0,C 180,E1 -4666.835,E2 -4666.835} C_VEL
LIN {X 0,Y 524.199,Z 384.723,A -85,B 0,C 180,E1 -4668.159,E2 -4668.159} C_VEL
LIN {X 0,Y 524.016,Z 392.756,A -85,B 0,C 180,E1 -4669.373,E2 -4669.373} C_VEL
LIN {X 0,Y 523.729,Z 400.311,A -85,B 0,C 180,E1 -4670.733,E2 -4670.733} C_VEL
LIN {X 0,Y 523.638,Z 405.746,A -85,B 0,C 180,E1 -4671.898,E2 -4671.898} C_VEL
LIN {X 0,Y 523.484,Z 411.701,A -85,B 0,C 180,E1 -4673.455,E2 -4673.455} C_VEL
LIN {X 0,Y 523.445,Z 415.15,A -85,B 0,C 180,E1 -4674.607,E2 -4674.607} C_VEL
LIN {X 0,Y 523.404,Z 418.71,A -85,B 0,C 180,E1 -4676.15,E2 -4676.15} C_VEL
LIN {X 0,Y 523.335,Z 421.041,A -85,B 0,C 180,E1 -4677.691,E2 -4677.691} C_VEL
LIN {X 0,Y 523.264,Z 422.214,A -85,B 0,C 180,E1 -4679.23,E2 -4679.23} C_VEL
LIN {X 0,Y 523.266,Z 422.26,A -85,B 0,C 180,E1 -4680.769,E2 -4680.769} C_VEL
LIN {X 0,Y 523.336,Z 421.178,A -85,B 0,C 180,E1 -4682.309,E2 -4682.309} C_VEL
LIN {X 0,Y 523.406,Z 418.952,A -85,B 0,C 180,E1 -4683.849,E2 -4683.849} C_VEL
LIN {X 0,Y 523.446,Z 415.499,A -85,B 0,C 180,E1 -4685.393,E2 -4685.393} C_VEL
LIN {X 0,Y 523.552,Z 410.749,A -85,B 0,C 180,E1 -4686.939,E2 -4686.939} C_VEL
LIN {X 0,Y 523.695,Z 404.626,A -85,B 0,C 180,E1 -4688.489,E2 -4688.489} C_VEL
LIN {X 0,Y 523.84,Z 396.862,A -85,B 0,C 180,E1 -4690.044,E2 -4690.044} C_VEL
LIN {X 0,Y 524.082,Z 388.536,A -85,B 0,C 180,E1 -4691.408,E2 -4691.408} C_VEL
LIN {X 0,Y 524.384,Z 380.044,A -85,B 0,C 180,E1 -4692.579,E2 -4692.579} C_VEL
LIN {X 0,Y 524.754,Z 369.969,A -85,B 0,C 180,E1 -4693.752,E2 -4693.752} C_VEL
LIN {X 0,Y 525.118,Z 359,A -85,B 0,C 180,E1 -4694.83,E2 -4694.83} C_VEL
LIN {X 0,Y 525.515,Z 347.567,A -85,B 0,C 180,E1 -4695.777,E2 -4695.777} C_VEL
LIN {X 0,Y 525.895,Z 334.202,A -85,B 0,C 180,E1 -4696.698,E2 -4696.698} C_VEL
LIN {X 0,Y 526.299,Z 319.995,A -85,B 0,C 180,E1 -4697.485,E2 -4697.485} C_VEL
LIN {X 0,Y 526.672,Z 305.437,A -85,B 0,C 180,E1 -4698.115,E2 -4698.115} C_VEL
LIN {X 0,Y 526.93,Z 290.366,A -85,B 0,C 180,E1 -4698.602,E2 -4698.602} C_VEL
LIN {X 0,Y 527.109,Z 275.153,A -85,B 0,C 180,E1 -4698.935,E2 -4698.935} C_VEL
LIN {X 0,Y 528.299,Z 149.749,A -85,B 0,C 180,E1 -4700.816,E2 -4700.816} C_VEL
LIN {X 0,Y 528.384,Z 125.15,A -85,B 0,C 180,E1 -4701.212,E2 -4701.212} C_VEL
LIN {X 0,Y 526.014,Z 115.631,A -85,B 0,C 180,E1 -4701.488,E2 -4701.488} C_VEL
LIN {X 0,Y 523.928,Z 105.85,A -85,B 0,C 180,E1 -4703.363,E2 -4703.363} C_VEL
LIN {X 0,Y 523.926,Z 105.85,A -85,B 0,C 180,E1 -4706.274,E2 -4706.274} C_VEL
LIN {X 0,Y 523.936,Z 105.849,A -85,B 0,C 180,E1 -4709.32,E2 -4709.32} C_VEL
LIN {X 0,Y 523.934,Z 105.845,A -85,B 0,C 180,E1 -4712.32,E2 -4712.32} C_VEL
LIN {X 0,Y 523.913,Z 105.851,A -85,B 0,C 180,E1 -4715.227,E2 -4715.227} C_VEL
LIN {X 0,Y 523.911,Z 105.848,A -85,B 0,C 180,E1 -4718.102,E2 -4718.102} C_VEL
LIN {X 0,Y 523.919,Z 105.852,A -85,B 0,C 180,E1 -4721.306,E2 -4721.306} C_VEL
LIN {X 0,Y 523.933,Z 105.846,A -85,B 0,C 180,E1 -4724.689,E2 -4724.689} C_VEL
LIN {X 0,Y 523.898,Z 105.849,A -85,B 0,C 180,E1 -4727.876,E2 -4727.876} C_VEL
LIN {X 0,Y 523.91,Z 105.853,A -85,B 0,C 180,E1 -4731.081,E2 -4731.081} C_VEL
LIN {X 0,Y 523.877,Z 105.853,A -85,B 0,C 180,E1 -4733.823,E2 -4733.823} C_VEL
LIN {X 0,Y 523.91,Z 105.853,A -85,B 0,C 180,E1 -4736.633,E2 -4736.633} C_VEL
LIN {X 0,Y 523.905,Z 105.853,A -85,B 0,C 180,E1 -4739.352,E2 -4739.352} C_VEL
LIN {X 0,Y 523.924,Z 106.061,A -85,B 0,C 180,E1 -4740.866,E2 -4740.866} C_VEL
LIN {X 0,Y 526.751,Z 117.978,A -85,B 0,C 180,E1 -4742.593,E2 -4742.593} C_VEL
LIN {X 0,Y 526.348,Z 136.239,A -85,B 0,C 180,E1 -4744.89,E2 -4744.89} C_VEL
LIN {X 0,Y 525.649,Z 161.921,A -85,B 0,C 180,E1 -4748.015,E2 -4748.015} C_VEL
LIN {X 0,Y 525.562,Z 165.925,A -85,B 0,C 180,E1 -4748.495,E2 -4748.495} C_VEL
LIN {X 0,Y 528.345,Z 183.797,A -85,B 0,C 180,E1 -4748.906,E2 -4748.906} C_VEL
LIN {X 0,Y 527.208,Z 306.204,A -85,B 0,C 180,E1 -4750.728,E2 -4750.728} C_VEL
LIN {X 0,Y 526.954,Z 335.12,A -85,B 0,C 180,E1 -4751.168,E2 -4751.168} C_VEL
LIN {X 0,Y 526.691,Z 350.543,A -85,B 0,C 180,E1 -4751.554,E2 -4751.554} C_VEL
LIN {X 0,Y 526.354,Z 365.162,A -85,B 0,C 180,E1 -4752.068,E2 -4752.068} C_VEL
LIN {X 0,Y 525.956,Z 379.092,A -85,B 0,C 180,E1 -4752.704,E2 -4752.704} C_VEL
LIN {X 0,Y 525.523,Z 392.818,A -85,B 0,C 180,E1 -4753.49,E2 -4753.49} C_VEL
LIN {X 0,Y 525.131,Z 406.774,A -85,B 0,C 180,E1 -4754.475,E2 -4754.475} C_VEL
LIN {X 0,Y 524.72,Z 419.408,A -85,B 0,C 180,E1 -4755.554,E2 -4755.554} C_VEL
LIN {X 0,Y 524.342,Z 431.745,A -85,B 0,C 180,E1 -4756.829,E2 -4756.829} C_VEL
LIN {X 0,Y 524.023,Z 442.339,A -85,B 0,C 180,E1 -4758.144,E2 -4758.144} C_VEL
LIN {X 0,Y 523.83,Z 451.839,A -85,B 0,C 180,E1 -4759.565,E2 -4759.565} C_VEL
LIN {X 0,Y 523.623,Z 458.39,A -85,B 0,C 180,E1 -4760.731,E2 -4760.731} C_VEL
LIN {X 0,Y 523.496,Z 465.597,A -85,B 0,C 180,E1 -4762.285,E2 -4762.285} C_VEL
LIN {X 0,Y 523.441,Z 471.248,A -85,B 0,C 180,E1 -4763.834,E2 -4763.834} C_VEL
LIN {X 0,Y 523.324,Z 475.513,A -85,B 0,C 180,E1 -4765.378,E2 -4765.378} C_VEL
LIN {X 0,Y 523.358,Z 478.508,A -85,B 0,C 180,E1 -4766.921,E2 -4766.921} C_VEL
LIN {X 0,Y 523.272,Z 480.289,A -85,B 0,C 180,E1 -4768.461,E2 -4768.461} C_VEL
LIN {X 0,Y 523.254,Z 480.905,A -85,B 0,C 180,E1 -4770,E2 -4770} C_VEL
LIN {X 0,Y 523.272,Z 480.304,A -85,B 0,C 180,E1 -4771.539,E2 -4771.539} C_VEL
LIN {X 0,Y 523.358,Z 478.545,A -85,B 0,C 180,E1 -4773.079,E2 -4773.079} C_VEL
LIN {X 0,Y 523.323,Z 475.583,A -85,B 0,C 180,E1 -4774.622,E2 -4774.622} C_VEL
LIN {X 0,Y 523.446,Z 471.362,A -85,B 0,C 180,E1 -4776.166,E2 -4776.166} C_VEL
LIN {X 0,Y 523.496,Z 465.751,A -85,B 0,C 180,E1 -4777.715,E2 -4777.715} C_VEL
LIN {X 0,Y 523.624,Z 458.606,A -85,B 0,C 180,E1 -4779.269,E2 -4779.269} C_VEL
LIN {X 0,Y 523.86,Z 450.959,A -85,B 0,C 180,E1 -4780.63,E2 -4780.63} C_VEL
LIN {X 0,Y 524.05,Z 442.009,A -85,B 0,C 180,E1 -4781.958,E2 -4781.958} C_VEL
LIN {X 0,Y 524.42,Z 430.572,A -85,B 0,C 180,E1 -4783.366,E2 -4783.366} C_VEL
LIN {X 0,Y 524.821,Z 419.101,A -85,B 0,C 180,E1 -4784.542,E2 -4784.542} C_VEL
LIN {X 0,Y 525.261,Z 406.486,A -85,B 0,C 180,E1 -4785.621,E2 -4785.621} C_VEL
LIN {X 0,Y 525.608,Z 394.076,A -85,B 0,C 180,E1 -4786.507,E2 -4786.507} C_VEL
LIN {X 0,Y 526.059,Z 380.668,A -85,B 0,C 180,E1 -4787.293,E2 -4787.293} C_VEL
LIN {X 0,Y 526.516,Z 366.021,A -85,B 0,C 180,E1 -4787.979,E2 -4787.979} C_VEL
LIN {X 0,Y 526.882,Z 350.199,A -85,B 0,C 180,E1 -4788.539,E2 -4788.539} C_VEL
LIN {X 0,Y 527.172,Z 335.063,A -85,B 0,C 180,E1 -4788.91,E2 -4788.91} C_VEL
LIN {X 0,Y 527.828,Z 256.274,A -85,B 0,C 180,E1 -4790.077,E2 -4790.077} C_VEL
LIN {X 0,Y 528.308,Z 191.784,A -85,B 0,C 180,E1 -4790.999,E2 -4790.999} C_VEL
LIN {X 0,Y 528.288,Z 178.529,A -85,B 0,C 180,E1 -4791.209,E2 -4791.209} C_VEL
LIN {X 0,Y 526.459,Z 165.958,A -85,B 0,C 180,E1 -4791.496,E2 -4791.496} C_VEL
LIN {X 0,Y 527.185,Z 137.649,A -85,B 0,C 180,E1 -4794.201,E2 -4794.201} C_VEL
LIN {X 0,Y 527.77,Z 120.509,A -85,B 0,C 180,E1 -4795.856,E2 -4795.856} C_VEL
LIN {X 0,Y 523.926,Z 105.851,A -85,B 0,C 180,E1 -4797.524,E2 -4797.524} C_VEL
LIN {X 0,Y 523.937,Z 105.847,A -85,B 0,C 180,E1 -4800.646,E2 -4800.646} C_VEL
LIN {X 0,Y 523.925,Z 105.845,A -85,B 0,C 180,E1 -4803.729,E2 -4803.729} C_VEL
LIN {X 0,Y 523.896,Z 105.85,A -85,B 0,C 180,E1 -4806.4,E2 -4806.4} C_VEL
LIN {X 0,Y 523.911,Z 105.853,A -85,B 0,C 180,E1 -4809.086,E2 -4809.086} C_VEL
LIN {X 0,Y 523.898,Z 105.848,A -85,B 0,C 180,E1 -4812.124,E2 -4812.124} C_VEL
LIN {X 0,Y 523.933,Z 105.843,A -85,B 0,C 180,E1 -4815.311,E2 -4815.311} C_VEL
LIN {X 0,Y 523.919,Z 105.85,A -85,B 0,C 180,E1 -4818.694,E2 -4818.694} C_VEL
LIN {X 0,Y 523.911,Z 105.848,A -85,B 0,C 180,E1 -4821.898,E2 -4821.898} C_VEL
LIN {X 0,Y 523.917,Z 105.849,A -85,B 0,C 180,E1 -4824.913,E2 -4824.913} C_VEL
LIN {X 0,Y 523.933,Z 105.845,A -85,B 0,C 180,E1 -4827.68,E2 -4827.68} C_VEL
LIN {X 0,Y 523.935,Z 105.849,A -85,B 0,C 180,E1 -4830.68,E2 -4830.68} C_VEL
LIN {X 0,Y 523.903,Z 105.851,A -85,B 0,C 180,E1 -4833.725,E2 -4833.725} C_VEL
LIN {X 0,Y 523.908,Z 105.854,A -85,B 0,C 180,E1 -4836.27,E2 -4836.27} C_VEL
LIN {X 0,Y 523.96,Z 105.982,A -85,B 0,C 180,E1 -4837.271,E2 -4837.271} C_VEL
LIN {X 0,Y 525.796,Z 114.646,A -85,B 0,C 180,E1 -4838.604,E2 -4838.604} C_VEL
LIN {X 0,Y 528.444,Z 125.679,A -85,B 0,C 180,E1 -4838.906,E2 -4838.906} C_VEL
LIN {X 0,Y 527.439,Z 229.532,A -85,B 0,C 180,E1 -4840.491,E2 -4840.491} C_VEL
LIN {X 0,Y 527.05,Z 279.249,A -85,B 0,C 180,E1 -4841.236,E2 -4841.236} C_VEL
LIN {X 0,Y 526.856,Z 294.574,A -85,B 0,C 180,E1 -4841.614,E2 -4841.614} C_VEL
LIN {X 0,Y 526.53,Z 309.058,A -85,B 0,C 180,E1 -4842.122,E2 -4842.122} C_VEL
LIN {X 0,Y 526.263,Z 321.994,A -85,B 0,C 180,E1 -4842.714,E2 -4842.714} C_VEL
LIN {X 0,Y 525.857,Z 335.78,A -85,B 0,C 180,E1 -4843.501,E2 -4843.501} C_VEL
LIN {X 0,Y 525.457,Z 348.171,A -85,B 0,C 180,E1 -4844.366,E2 -4844.366} C_VEL
LIN {X 0,Y 525.05,Z 360.087,A -85,B 0,C 180,E1 -4845.366,E2 -4845.366} C_VEL
LIN {X 0,Y 524.717,Z 370.877,A -85,B 0,C 180,E1 -4846.444,E2 -4846.444} C_VEL
LIN {X 0,Y 524.357,Z 380.805,A -85,B 0,C 180,E1 -4847.617,E2 -4847.617} C_VEL
LIN {X 0,Y 524.106,Z 390.448,A -85,B 0,C 180,E1 -4848.984,E2 -4848.984} C_VEL
LIN {X 0,Y 523.817,Z 398.452,A -85,B 0,C 180,E1 -4850.345,E2 -4850.345} C_VEL
LIN {X 0,Y 523.639,Z 405.881,A -85,B 0,C 180,E1 -4851.899,E2 -4851.899} C_VEL
LIN {X 0,Y 523.49,Z 411.768,A -85,B 0,C 180,E1 -4853.449,E2 -4853.449} C_VEL
LIN {X 0,Y 523.446,Z 415.21,A -85,B 0,C 180,E1 -4854.607,E2 -4854.607} C_VEL
LIN {X 0,Y 523.404,Z 418.732,A -85,B 0,C 180,E1 -4856.151,E2 -4856.151} C_VEL
LIN {X 0,Y 523.335,Z 421.057,A -85,B 0,C 180,E1 -4857.691,E2 -4857.691} C_VEL
LIN {X 0,Y 523.264,Z 422.238,A -85,B 0,C 180,E1 -4859.231,E2 -4859.231} C_VEL
LIN {X 0,Y 523.263,Z 422.243,A -85,B 0,C 180,E1 -4860.77,E2 -4860.77} C_VEL
LIN {X 0,Y 523.336,Z 421.109,A -85,B 0,C 180,E1 -4862.309,E2 -4862.309} C_VEL
LIN {X 0,Y 523.404,Z 418.831,A -85,B 0,C 180,E1 -4863.85,E2 -4863.85} C_VEL
LIN {X 0,Y 523.445,Z 415.354,A -85,B 0,C 180,E1 -4865.393,E2 -4865.393} C_VEL
LIN {X 0,Y 523.543,Z 410.591,A -85,B 0,C 180,E1 -4866.939,E2 -4866.939} C_VEL
LIN {X 0,Y 523.652,Z 404.416,A -85,B 0,C 180,E1 -4868.49,E2 -4868.49} C_VEL
LIN {X 0,Y 523.825,Z 396.632,A -85,B 0,C 180,E1 -4870.045,E2 -4870.045} C_VEL
LIN {X 0,Y 524.074,Z 388.3,A -85,B 0,C 180,E1 -4871.409,E2 -4871.409} C_VEL
LIN {X 0,Y 524.453,Z 378.242,A -85,B 0,C 180,E1 -4872.775,E2 -4872.775} C_VEL
LIN {X 0,Y 524.793,Z 367.929,A -85,B 0,C 180,E1 -4873.949,E2 -4873.949} C_VEL
LIN {X 0,Y 525.166,Z 356.742,A -85,B 0,C 180,E1 -4875.024,E2 -4875.024} C_VEL
LIN {X 0,Y 525.632,Z 344.509,A -85,B 0,C 180,E1 -4876.008,E2 -4876.008} C_VEL
LIN {X 0,Y 526.032,Z 331.196,A -85,B 0,C 180,E1 -4876.894,E2 -4876.894} C_VEL
LIN {X 0,Y 526.457,Z 316.404,A -85,B 0,C 180,E1 -4877.681,E2 -4877.681} C_VEL
LIN {X 0,Y 526.83,Z 301.535,A -85,B 0,C 180,E1 -4878.292,E2 -4878.292} C_VEL
LIN {X 0,Y 527.088,Z 286.861,A -85,B 0,C 180,E1 -4878.739,E2 -4878.739} C_VEL
LIN {X 0,Y 527.266,Z 270.942,A -85,B 0,C 180,E1 -4879.06,E2 -4879.06} C_VEL
LIN {X 0,Y 528.551,Z 126.541,A -85,B 0,C 180,E1 -4881.171,E2 -4881.171} C_VEL
LIN {X 0,Y 525.457,Z 113.218,A -85,B 0,C 180,E1 -4881.507,E2 -4881.507} C_VEL
LIN {X 0,Y 523.924,Z 105.849,A -85,B 0,C 180,E1 -4882.727,E2 -4882.727} C_VEL
LIN {X 0,Y 523.906,Z 105.851,A -85,B 0,C 180,E1 -4885.574,E2 -4885.574} C_VEL
LIN {X 0,Y 523.238,Z 105.934,A -85,B 0,C 180,E1 -4886.216,E2 -4886.216} C_VEL
LIN {X 0,Y 520.362,Z 106.29,A -85,B 0,C 180,E1 -4887.258,E2 -4887.258} C_VEL
LIN {X 0,Y 517.947,Z 106.593,A -85,B 0,C 180,E1 -4888.098,E2 -4888.098} C_VEL
LIN {X 0,Y 516.938,Z 106.715,A -85,B 0,C 180,E1 -4888.746,E2 -4888.746} C_VEL
LIN {X 0,Y 516.871,Z 106.723,A -85,B 0,C 180,E1 -4888.966,E2 -4888.966} C_VEL
LIN {X 0,Y 516.874,Z 106.726,A -85,B 0,C 180,E1 -4892.025,E2 -4892.025} C_VEL
LIN {X 0,Y 516.875,Z 106.722,A -85,B 0,C 180,E1 -4894.826,E2 -4894.826} C_VEL
LIN {X 0,Y 516.879,Z 106.724,A -85,B 0,C 180,E1 -4897.943,E2 -4897.943} C_VEL
LIN {X 0,Y 516.855,Z 106.725,A -85,B 0,C 180,E1 -4900.745,E2 -4900.745} C_VEL
LIN {X 0,Y 516.883,Z 106.72,A -85,B 0,C 180,E1 -4903.904,E2 -4903.904} C_VEL
LIN {X 0,Y 516.882,Z 106.711,A -85,B 0,C 180,E1 -4906.108,E2 -4906.108} C_VEL
LIN {X 0,Y 516.855,Z 106.73,A -85,B 0,C 180,E1 -4909.255,E2 -4909.255} C_VEL
LIN {X 0,Y 516.862,Z 106.722,A -85,B 0,C 180,E1 -4912.274,E2 -4912.274} C_VEL
LIN {X 0,Y 516.875,Z 106.724,A -85,B 0,C 180,E1 -4915.175,E2 -4915.175} C_VEL
LIN {X 0,Y 516.868,Z 106.722,A -85,B 0,C 180,E1 -4917.975,E2 -4917.975} C_VEL
LIN {X 0,Y 516.901,Z 106.719,A -85,B 0,C 180,E1 -4920.694,E2 -4920.694} C_VEL
LIN {X 0,Y 516.884,Z 106.721,A -85,B 0,C 180,E1 -4923.818,E2 -4923.818} C_VEL
LIN {X 0,Y 516.845,Z 106.73,A -85,B 0,C 180,E1 -4926.775,E2 -4926.775} C_VEL
LIN {X 0,Y 516.91,Z 106.715,A -85,B 0,C 180,E1 -4929.742,E2 -4929.742} C_VEL
LIN {X 0,Y 516.882,Z 106.728,A -85,B 0,C 180,E1 -4932.594,E2 -4932.594} C_VEL
LIN {X 0,Y 516.933,Z 106.718,A -85,B 0,C 180,E1 -4935.03,E2 -4935.03} C_VEL
LIN {X 0,Y 516.971,Z 106.715,A -85,B 0,C 180,E1 -4938.234,E2 -4938.234} C_VEL
LIN {X 0,Y 516.923,Z 106.716,A -85,B 0,C 180,E1 -4941.399,E2 -4941.399} C_VEL
LIN {X 0,Y 516.981,Z 106.715,A -85,B 0,C 180,E1 -4944.539,E2 -4944.539} C_VEL
LIN {X 0,Y 517.075,Z 106.702,A -85,B 0,C 180,E1 -4947.663,E2 -4947.663} C_VEL
LIN {X 0,Y 516.933,Z 106.721,A -85,B 0,C 180,E1 -4950.389,E2 -4950.389} C_VEL
LIN {X 0,Y 516.955,Z 107,A -85,B 0,C 180,E1 -4950.536,E2 -4950.536} C_VEL
LIN {X 0,Y 519.341,Z 117.925,A -85,B 0,C 180,E1 -4952.133,E2 -4952.133} C_VEL
LIN {X 0,Y 519.186,Z 133.768,A -85,B 0,C 180,E1 -4954.27,E2 -4954.27} C_VEL
LIN {X 0,Y 518.943,Z 141.23,A -85,B 0,C 180,E1 -4955.269,E2 -4955.269} C_VEL
LIN {X 0,Y 521.885,Z 154.522,A -85,B 0,C 180,E1 -4955.603,E2 -4955.603} C_VEL
LIN {X 0,Y 520.805,Z 306.927,A -85,B 0,C 180,E1 -4957.78,E2 -4957.78} C_VEL
LIN {X 0,Y 520.551,Z 322.149,A -85,B 0,C 180,E1 -4958.15,E2 -4958.15} C_VEL
LIN {X 0,Y 520.167,Z 337.145,A -85,B 0,C 180,E1 -4958.675,E2 -4958.675} C_VEL
LIN {X 0,Y 519.724,Z 351.41,A -85,B 0,C 180,E1 -4959.339,E2 -4959.339} C_VEL
LIN {X 0,Y 519.223,Z 364.983,A -85,B 0,C 180,E1 -4960.135,E2 -4960.135} C_VEL
LIN {X 0,Y 518.721,Z 377.541,A -85,B 0,C 180,E1 -4961.033,E2 -4961.033} C_VEL
LIN {X 0,Y 518.204,Z 390.215,A -85,B 0,C 180,E1 -4962.133,E2 -4962.133} C_VEL
LIN {X 0,Y 517.718,Z 401.779,A -85,B 0,C 180,E1 -4963.343,E2 -4963.343} C_VEL
LIN {X 0,Y 517.305,Z 411.595,A -85,B 0,C 180,E1 -4964.557,E2 -4964.557} C_VEL
LIN {X 0,Y 516.949,Z 421.204,A -85,B 0,C 180,E1 -4965.98,E2 -4965.98} C_VEL
LIN {X 0,Y 516.69,Z 429.175,A -85,B 0,C 180,E1 -4967.412,E2 -4967.412} C_VEL
LIN {X 0,Y 516.546,Z 434.939,A -85,B 0,C 180,E1 -4968.647,E2 -4968.647} C_VEL
LIN {X 0,Y 516.423,Z 440.527,A -85,B 0,C 180,E1 -4970.111,E2 -4970.111} C_VEL
LIN {X 0,Y 516.348,Z 444.928,A -85,B 0,C 180,E1 -4971.561,E2 -4971.561} C_VEL
LIN {X 0,Y 516.186,Z 448.682,A -85,B 0,C 180,E1 -4973.256,E2 -4973.256} C_VEL
LIN {X 0,Y 516.154,Z 450.996,A -85,B 0,C 180,E1 -4974.967,E2 -4974.967} C_VEL
LIN {X 0,Y 516.156,Z 451.784,A -85,B 0,C 180,E1 -4976.017,E2 -4976.017} C_VEL
LIN {X 0,Y 516.177,Z 451.884,A -85,B 0,C 180,E1 -4977.747,E2 -4977.747} C_VEL
LIN {X 0,Y 516.225,Z 450.746,A -85,B 0,C 180,E1 -4979.388,E2 -4979.388} C_VEL
LIN {X 0,Y 516.237,Z 448.102,A -85,B 0,C 180,E1 -4981.153,E2 -4981.153} C_VEL
LIN {X 0,Y 516.319,Z 445.176,A -85,B 0,C 180,E1 -4982.442,E2 -4982.442} C_VEL
LIN {X 0,Y 516.39,Z 440.766,A -85,B 0,C 180,E1 -4983.918,E2 -4983.918} C_VEL
LIN {X 0,Y 516.552,Z 434.699,A -85,B 0,C 180,E1 -4985.508,E2 -4985.508} C_VEL
LIN {X 0,Y 516.759,Z 427.577,A -85,B 0,C 180,E1 -4986.999,E2 -4986.999} C_VEL
LIN {X 0,Y 517.048,Z 418.794,A -85,B 0,C 180,E1 -4988.494,E2 -4988.494} C_VEL
LIN {X 0,Y 517.323,Z 410.535,A -85,B 0,C 180,E1 -4989.681,E2 -4989.681} C_VEL
LIN {X 0,Y 517.77,Z 400.396,A -85,B 0,C 180,E1 -4990.914,E2 -4990.914} C_VEL
LIN {X 0,Y 518.285,Z 388.061,A -85,B 0,C 180,E1 -4992.165,E2 -4992.165} C_VEL
LIN {X 0,Y 518.772,Z 376.073,A -85,B 0,C 180,E1 -4993.175,E2 -4993.175} C_VEL
LIN {X 0,Y 519.286,Z 363.516,A -85,B 0,C 180,E1 -4994.056,E2 -4994.056} C_VEL
LIN {X 0,Y 519.793,Z 349.357,A -85,B 0,C 180,E1 -4994.862,E2 -4994.862} C_VEL
LIN {X 0,Y 520.247,Z 334.401,A -85,B 0,C 180,E1 -4995.525,E2 -4995.525} C_VEL
LIN {X 0,Y 520.611,Z 318.988,A -85,B 0,C 180,E1 -4996.029,E2 -4996.029} C_VEL
LIN {X 0,Y 520.809,Z 304.335,A -85,B 0,C 180,E1 -4996.356,E2 -4996.356} C_VEL
LIN {X 0,Y 521.921,Z 151.84,A -85,B 0,C 180,E1 -4998.524,E2 -4998.524} C_VEL
LIN {X 0,Y 519.75,Z 139.695,A -85,B 0,C 180,E1 -4998.811,E2 -4998.811} C_VEL
LIN {X 0,Y 520.148,Z 120.317,A -85,B 0,C 180,E1 -5000.827,E2 -5000.827} C_VEL
LIN {X 0,Y 516.891,Z 106.727,A -85,B 0,C 180,E1 -5002.43,E2 -5002.43} C_VEL
LIN {X 0,Y 516.885,Z 106.723,A -85,B 0,C 180,E1 -5005.175,E2 -5005.175} C_VEL
LIN {X 0,Y 516.877,Z 106.728,A -85,B 0,C 180,E1 -5007.975,E2 -5007.975} C_VEL
LIN {X 0,Y 516.925,Z 106.715,A -85,B 0,C 180,E1 -5010.695,E2 -5010.695} C_VEL
LIN {X 0,Y 516.945,Z 106.719,A -85,B 0,C 180,E1 -5013.804,E2 -5013.804} C_VEL
LIN {X 0,Y 516.868,Z 106.729,A -85,B 0,C 180,E1 -5016.776,E2 -5016.776} C_VEL
LIN {X 0,Y 516.899,Z 106.771,A -85,B 0,C 180,E1 -5017.481,E2 -5017.481} C_VEL
LIN {X 0,Y 518.183,Z 112.212,A -85,B 0,C 180,E1 -5018.238,E2 -5018.238} C_VEL
LIN {X 0,Y 521.407,Z 121.139,A -85,B 0,C 180,E1 -5018.523,E2 -5018.523} C_VEL
LIN {X 0,Y 521.93,Z 124.366,A -85,B 0,C 180,E1 -5018.597,E2 -5018.597} C_VEL
LIN {X 0,Y 520.458,Z 279.42,A -85,B 0,C 180,E1 -5020.942,E2 -5020.942} C_VEL
LIN {X 0,Y 520.214,Z 294.543,A -85,B 0,C 180,E1 -5021.327,E2 -5021.327} C_VEL
LIN {X 0,Y 519.842,Z 309.843,A -85,B 0,C 180,E1 -5021.883,E2 -5021.883} C_VEL
LIN {X 0,Y 519.444,Z 324.36,A -85,B 0,C 180,E1 -5022.581,E2 -5022.581} C_VEL
LIN {X 0,Y 518.979,Z 337.617,A -85,B 0,C 180,E1 -5023.377,E2 -5023.377} C_VEL
LIN {X 0,Y 518.526,Z 351.164,A -85,B 0,C 180,E1 -5024.378,E2 -5024.378} C_VEL
LIN {X 0,Y 518.036,Z 363.321,A -85,B 0,C 180,E1 -5025.464,E2 -5025.464} C_VEL
LIN {X 0,Y 517.635,Z 374.455,A -85,B 0,C 180,E1 -5026.655,E2 -5026.655} C_VEL
LIN {X 0,Y 517.293,Z 383.826,A -85,B 0,C 180,E1 -5027.843,E2 -5027.843} C_VEL
LIN {X 0,Y 517.019,Z 392.993,A -85,B 0,C 180,E1 -5029.227,E2 -5029.227} C_VEL
LIN {X 0,Y 516.711,Z 400.58,A -85,B 0,C 180,E1 -5030.606,E2 -5030.606} C_VEL
LIN {X 0,Y 516.526,Z 407.668,A -85,B 0,C 180,E1 -5032.18,E2 -5032.18} C_VEL
LIN {X 0,Y 516.422,Z 413.236,A -85,B 0,C 180,E1 -5033.749,E2 -5033.749} C_VEL
LIN {X 0,Y 516.275,Z 417.429,A -85,B 0,C 180,E1 -5035.315,E2 -5035.315} C_VEL
LIN {X 0,Y 516.372,Z 420.377,A -85,B 0,C 180,E1 -5036.879,E2 -5036.879} C_VEL
LIN {X 0,Y 516.192,Z 422.185,A -85,B 0,C 180,E1 -5038.439,E2 -5038.439} C_VEL
LIN {X 0,Y 516.177,Z 422.818,A -85,B 0,C 180,E1 -5040,E2 -5040} C_VEL
LIN {X 0,Y 516.194,Z 422.288,A -85,B 0,C 180,E1 -5041.56,E2 -5041.56} C_VEL
LIN {X 0,Y 516.373,Z 420.597,A -85,B 0,C 180,E1 -5043.121,E2 -5043.121} C_VEL
LIN {X 0,Y 516.293,Z 417.755,A -85,B 0,C 180,E1 -5044.685,E2 -5044.685} C_VEL
LIN {X 0,Y 516.473,Z 413.666,A -85,B 0,C 180,E1 -5046.249,E2 -5046.249} C_VEL
LIN {X 0,Y 516.554,Z 408.22,A -85,B 0,C 180,E1 -5047.819,E2 -5047.819} C_VEL
LIN {X 0,Y 516.708,Z 401.26,A -85,B 0,C 180,E1 -5049.393,E2 -5049.393} C_VEL
LIN {X 0,Y 517.005,Z 393.765,A -85,B 0,C 180,E1 -5050.772,E2 -5050.772} C_VEL
LIN {X 0,Y 517.254,Z 384.977,A -85,B 0,C 180,E1 -5052.118,E2 -5052.118} C_VEL
LIN {X 0,Y 517.631,Z 375.377,A -85,B 0,C 180,E1 -5053.345,E2 -5053.345} C_VEL
LIN {X 0,Y 518.059,Z 363.32,A -85,B 0,C 180,E1 -5054.635,E2 -5054.635} C_VEL
LIN {X 0,Y 518.531,Z 350.934,A -85,B 0,C 180,E1 -5055.728,E2 -5055.728} C_VEL
LIN {X 0,Y 518.918,Z 338.695,A -85,B 0,C 180,E1 -5056.625,E2 -5056.625} C_VEL
LIN {X 0,Y 519.369,Z 325.466,A -85,B 0,C 180,E1 -5057.421,E2 -5057.421} C_VEL
LIN {X 0,Y 519.708,Z 312.063,A -85,B 0,C 180,E1 -5058.07,E2 -5058.07} C_VEL
LIN {X 0,Y 519.998,Z 297.711,A -85,B 0,C 180,E1 -5058.609,E2 -5058.609} C_VEL
LIN {X 0,Y 520.192,Z 282.889,A -85,B 0,C 180,E1 -5059.012,E2 -5059.012} C_VEL
LIN {X 0,Y 520.392,Z 261.403,A -85,B 0,C 180,E1 -5059.373,E2 -5059.373} C_VEL
LIN {X 0,Y 521.675,Z 151.264,A -85,B 0,C 180,E1 -5061.073,E2 -5061.073} C_VEL
LIN {X 0,Y 521.885,Z 126.564,A -85,B 0,C 180,E1 -5061.484,E2 -5061.484} C_VEL
LIN {X 0,Y 519.176,Z 116.706,A -85,B 0,C 180,E1 -5061.778,E2 -5061.778} C_VEL
LIN {X 0,Y 518.994,Z 115.954,A -85,B 0,C 180,E1 -5061.863,E2 -5061.863} C_VEL
LIN {X 0,Y 516.88,Z 106.729,A -85,B 0,C 180,E1 -5063.674,E2 -5063.674} C_VEL
LIN {X 0,Y 516.888,Z 106.725,A -85,B 0,C 180,E1 -5066.66,E2 -5066.66} C_VEL
LIN {X 0,Y 516.886,Z 106.728,A -85,B 0,C 180,E1 -5069.518,E2 -5069.518} C_VEL
LIN {X 0,Y 516.893,Z 106.722,A -85,B 0,C 180,E1 -5072.543,E2 -5072.543} C_VEL
LIN {X 0,Y 516.859,Z 106.73,A -85,B 0,C 180,E1 -5075.328,E2 -5075.328} C_VEL
LIN {X 0,Y 516.877,Z 106.726,A -85,B 0,C 180,E1 -5077.942,E2 -5077.942} C_VEL
LIN {X 0,Y 516.852,Z 106.727,A -85,B 0,C 180,E1 -5080.745,E2 -5080.745} C_VEL
LIN {X 0,Y 516.879,Z 106.724,A -85,B 0,C 180,E1 -5083.903,E2 -5083.903} C_VEL
LIN {X 0,Y 516.879,Z 106.723,A -85,B 0,C 180,E1 -5086.107,E2 -5086.107} C_VEL
LIN {X 0,Y 516.851,Z 106.732,A -85,B 0,C 180,E1 -5089.255,E2 -5089.255} C_VEL
LIN {X 0,Y 516.858,Z 106.727,A -85,B 0,C 180,E1 -5092.274,E2 -5092.274} C_VEL
LIN {X 0,Y 516.869,Z 106.73,A -85,B 0,C 180,E1 -5095.174,E2 -5095.174} C_VEL
LIN {X 0,Y 516.864,Z 106.728,A -85,B 0,C 180,E1 -5097.974,E2 -5097.974} C_VEL
LIN {X 0,Y 516.831,Z 106.798,A -85,B 0,C 180,E1 -5100.524,E2 -5100.524} C_VEL
LIN {X 0,Y 519.925,Z 119.5,A -85,B 0,C 180,E1 -5102.421,E2 -5102.421} C_VEL
LIN {X 0,Y 519.773,Z 129.45,A -85,B 0,C 180,E1 -5103.716,E2 -5103.716} C_VEL
LIN {X 0,Y 519.035,Z 151.298,A -85,B 0,C 180,E1 -5106.456,E2 -5106.456} C_VEL
LIN {X 0,Y 518.672,Z 165.363,A -85,B 0,C 180,E1 -5108.184,E2 -5108.184} C_VEL
LIN {X 0,Y 521.704,Z 184.599,A -85,B 0,C 180,E1 -5108.645,E2 -5108.645} C_VEL
LIN {X 0,Y 520.477,Z 298.798,A -85,B 0,C 180,E1 -5110.399,E2 -5110.399} C_VEL
LIN {X 0,Y 520.134,Z 334.554,A -85,B 0,C 180,E1 -5110.95,E2 -5110.95} C_VEL
LIN {X 0,Y 519.838,Z 349.806,A -85,B 0,C 180,E1 -5111.334,E2 -5111.334} C_VEL
LIN {X 0,Y 519.45,Z 364.844,A -85,B 0,C 180,E1 -5111.869,E2 -5111.869} C_VEL
LIN {X 0,Y 519.008,Z 379.706,A -85,B 0,C 180,E1 -5112.566,E2 -5112.566} C_VEL
LIN {X 0,Y 518.56,Z 393.263,A -85,B 0,C 180,E1 -5113.363,E2 -5113.363} C_VEL
LIN {X 0,Y 518.173,Z 405.819,A -85,B 0,C 180,E1 -5114.261,E2 -5114.261} C_VEL
LIN {X 0,Y 517.723,Z 418.561,A -85,B 0,C 180,E1 -5115.355,E2 -5115.355} C_VEL
LIN {X 0,Y 517.308,Z 430.998,A -85,B 0,C 180,E1 -5116.647,E2 -5116.647} C_VEL
LIN {X 0,Y 517.031,Z 440.63,A -85,B 0,C 180,E1 -5117.837,E2 -5117.837} C_VEL
LIN {X 0,Y 516.763,Z 450.038,A -85,B 0,C 180,E1 -5119.222,E2 -5119.222} C_VEL
LIN {X 0,Y 516.537,Z 457.819,A -85,B 0,C 180,E1 -5120.603,E2 -5120.603} C_VEL
LIN {X 0,Y 516.434,Z 465.079,A -85,B 0,C 180,E1 -5122.179,E2 -5122.179} C_VEL
LIN {X 0,Y 516.36,Z 470.771,A -85,B 0,C 180,E1 -5123.749,E2 -5123.749} C_VEL
LIN {X 0,Y 516.374,Z 473.087,A -85,B 0,C 180,E1 -5124.533,E2 -5124.533} C_VEL
LIN {X 0,Y 516.325,Z 476.733,A -85,B 0,C 180,E1 -5126.098,E2 -5126.098} C_VEL
LIN {X 0,Y 516.258,Z 479.134,A -85,B 0,C 180,E1 -5127.659,E2 -5127.659} C_VEL
LIN {X 0,Y 516.163,Z 480.345,A -85,B 0,C 180,E1 -5129.22,E2 -5129.22} C_VEL
LIN {X 0,Y 516.162,Z 480.36,A -85,B 0,C 180,E1 -5130.78,E2 -5130.78} C_VEL
LIN {X 0,Y 516.258,Z 479.179,A -85,B 0,C 180,E1 -5132.341,E2 -5132.341} C_VEL
LIN {X 0,Y 516.325,Z 476.82,A -85,B 0,C 180,E1 -5133.902,E2 -5133.902} C_VEL
LIN {X 0,Y 516.374,Z 473.227,A -85,B 0,C 180,E1 -5135.467,E2 -5135.467} C_VEL
LIN {X 0,Y 516.395,Z 468.304,A -85,B 0,C 180,E1 -5137.036,E2 -5137.036} C_VEL
LIN {X 0,Y 516.498,Z 461.923,A -85,B 0,C 180,E1 -5138.608,E2 -5138.608} C_VEL
LIN {X 0,Y 516.679,Z 453.902,A -85,B 0,C 180,E1 -5140.185,E2 -5140.185} C_VEL
LIN {X 0,Y 516.872,Z 444.903,A -85,B 0,C 180,E1 -5141.633,E2 -5141.633} C_VEL
LIN {X 0,Y 517.209,Z 435.025,A -85,B 0,C 180,E1 -5142.956,E2 -5142.956} C_VEL
LIN {X 0,Y 517.574,Z 424.473,A -85,B 0,C 180,E1 -5144.147,E2 -5144.147} C_VEL
LIN {X 0,Y 517.997,Z 412.727,A -85,B 0,C 180,E1 -5145.264,E2 -5145.264} C_VEL
LIN {X 0,Y 518.468,Z 400.525,A -85,B 0,C 180,E1 -5146.235,E2 -5146.235} C_VEL
LIN {X 0,Y 518.999,Z 386.925,A -85,B 0,C 180,E1 -5147.129,E2 -5147.129} C_VEL
LIN {X 0,Y 519.428,Z 372.888,A -85,B 0,C 180,E1 -5147.877,E2 -5147.877} C_VEL
LIN {X 0,Y 519.878,Z 358.164,A -85,B 0,C 180,E1 -5148.488,E2 -5148.488} C_VEL
LIN {X 0,Y 520.23,Z 342.447,A -85,B 0,C 180,E1 -5148.968,E2 -5148.968} C_VEL
LIN {X 0,Y 520.463,Z 325.972,A -85,B 0,C 180,E1 -5149.291,E2 -5149.291} C_VEL
LIN {X 0,Y 521.275,Z 237.294,A -85,B 0,C 180,E1 -5150.593,E2 -5150.593} C_VEL
LIN {X 0,Y 521.69,Z 179.757,A -85,B 0,C 180,E1 -5151.466,E2 -5151.466} C_VEL
LIN {X 0,Y 519.624,Z 165.642,A -85,B 0,C 180,E1 -5151.794,E2 -5151.794} C_VEL
LIN {X 0,Y 520.416,Z 138.424,A -85,B 0,C 180,E1 -5154.43,E2 -5154.43} C_VEL
LIN {X 0,Y 521.023,Z 122.395,A -85,B 0,C 180,E1 -5156.001,E2 -5156.001} C_VEL
LIN {X 0,Y 516.885,Z 106.727,A -85,B 0,C 180,E1 -5157.816,E2 -5157.816} C_VEL
LIN {X 0,Y 516.862,Z 106.726,A -85,B 0,C 180,E1 -5160.206,E2 -5160.206} C_VEL
LIN {X 0,Y 516.878,Z 106.728,A -85,B 0,C 180,E1 -5162.948,E2 -5162.948} C_VEL
LIN {X 0,Y 516.865,Z 106.725,A -85,B 0,C 180,E1 -5165.781,E2 -5165.781} C_VEL
LIN {X 0,Y 516.875,Z 106.728,A -85,B 0,C 180,E1 -5168.717,E2 -5168.717} C_VEL
LIN {X 0,Y 516.849,Z 106.726,A -85,B 0,C 180,E1 -5171.782,E2 -5171.782} C_VEL
LIN {X 0,Y 516.895,Z 106.723,A -85,B 0,C 180,E1 -5175.007,E2 -5175.007} C_VEL
LIN {X 0,Y 516.855,Z 106.729,A -85,B 0,C 180,E1 -5178.406,E2 -5178.406} C_VEL
LIN {X 0,Y 516.875,Z 106.724,A -85,B 0,C 180,E1 -5181.284,E2 -5181.284} C_VEL
LIN {X 0,Y 516.865,Z 106.729,A -85,B 0,C 180,E1 -5184.219,E2 -5184.219} C_VEL
LIN {X 0,Y 516.88,Z 106.724,A -85,B 0,C 180,E1 -5187.052,E2 -5187.052} C_VEL
LIN {X 0,Y 516.866,Z 106.726,A -85,B 0,C 180,E1 -5189.795,E2 -5189.795} C_VEL
LIN {X 0,Y 516.876,Z 106.729,A -85,B 0,C 180,E1 -5192.465,E2 -5192.465} C_VEL
LIN {X 0,Y 516.845,Z 106.73,A -85,B 0,C 180,E1 -5195.069,E2 -5195.069} C_VEL
LIN {X 0,Y 516.902,Z 106.859,A -85,B 0,C 180,E1 -5197.002,E2 -5197.002} C_VEL
LIN {X 0,Y 518.679,Z 114.897,A -85,B 0,C 180,E1 -5198.268,E2 -5198.268} C_VEL
LIN {X 0,Y 520.748,Z 121.751,A -85,B 0,C 180,E1 -5198.495,E2 -5198.495} C_VEL
LIN {X 0,Y 521.884,Z 128.023,A -85,B 0,C 180,E1 -5198.653,E2 -5198.653} C_VEL
LIN {X 0,Y 520.669,Z 231.396,A -85,B 0,C 180,E1 -5200.279,E2 -5200.279} C_VEL
LIN {X 0,Y 520.255,Z 280.286,A -85,B 0,C 180,E1 -5201.032,E2 -5201.032} C_VEL
LIN {X 0,Y 520.026,Z 295.604,A -85,B 0,C 180,E1 -5201.422,E2 -5201.422} C_VEL
LIN {X 0,Y 519.707,Z 310.985,A -85,B 0,C 180,E1 -5201.981,E2 -5201.981} C_VEL
LIN {X 0,Y 519.326,Z 325.498,A -85,B 0,C 180,E1 -5202.679,E2 -5202.679} C_VEL
LIN {X 0,Y 518.913,Z 338.686,A -85,B 0,C 180,E1 -5203.476,E2 -5203.476} C_VEL
LIN {X 0,Y 518.469,Z 351.263,A -85,B 0,C 180,E1 -5204.401,E2 -5204.401} C_VEL
LIN {X 0,Y 518.018,Z 363.276,A -85,B 0,C 180,E1 -5205.464,E2 -5205.464} C_VEL
LIN {X 0,Y 517.631,Z 374.498,A -85,B 0,C 180,E1 -5206.655,E2 -5206.655} C_VEL
LIN {X 0,Y 517.293,Z 384.2,A -85,B 0,C 180,E1 -5207.883,E2 -5207.883} C_VEL
LIN {X 0,Y 517.018,Z 393.108,A -85,B 0,C 180,E1 -5209.228,E2 -5209.228} C_VEL
LIN {X 0,Y 516.72,Z 400.721,A -85,B 0,C 180,E1 -5210.607,E2 -5210.607} C_VEL
LIN {X 0,Y 516.557,Z 407.784,A -85,B 0,C 180,E1 -5212.181,E2 -5212.181} C_VEL
LIN {X 0,Y 516.475,Z 413.322,A -85,B 0,C 180,E1 -5213.751,E2 -5213.751} C_VEL
LIN {X 0,Y 516.276,Z 417.502,A -85,B 0,C 180,E1 -5215.315,E2 -5215.315} C_VEL
LIN {X 0,Y 516.371,Z 420.419,A -85,B 0,C 180,E1 -5216.879,E2 -5216.879} C_VEL
LIN {X 0,Y 516.192,Z 422.179,A -85,B 0,C 180,E1 -5218.44,E2 -5218.44} C_VEL
LIN {X 0,Y 516.174,Z 422.772,A -85,B 0,C 180,E1 -5220,E2 -5220} C_VEL
LIN {X 0,Y 516.193,Z 422.194,A -85,B 0,C 180,E1 -5221.561,E2 -5221.561} C_VEL
LIN {X 0,Y 516.373,Z 420.474,A -85,B 0,C 180,E1 -5223.121,E2 -5223.121} C_VEL
LIN {X 0,Y 516.269,Z 417.592,A -85,B 0,C 180,E1 -5224.685,E2 -5224.685} C_VEL
LIN {X 0,Y 516.415,Z 413.454,A -85,B 0,C 180,E1 -5226.251,E2 -5226.251} C_VEL
LIN {X 0,Y 516.524,Z 407.972,A -85,B 0,C 180,E1 -5227.82,E2 -5227.82} C_VEL
LIN {X 0,Y 516.698,Z 400.983,A -85,B 0,C 180,E1 -5229.394,E2 -5229.394} C_VEL
LIN {X 0,Y 516.979,Z 393.463,A -85,B 0,C 180,E1 -5230.774,E2 -5230.774} C_VEL
LIN {X 0,Y 517.223,Z 384.393,A -85,B 0,C 180,E1 -5232.158,E2 -5232.158} C_VEL
LIN {X 0,Y 517.593,Z 375.147,A -85,B 0,C 180,E1 -5233.346,E2 -5233.346} C_VEL
LIN {X 0,Y 517.997,Z 364.15,A -85,B 0,C 180,E1 -5234.537,E2 -5234.537} C_VEL
LIN {X 0,Y 518.431,Z 352.525,A -85,B 0,C 180,E1 -5235.593,E2 -5235.593} C_VEL
LIN {X 0,Y 518.931,Z 338.83,A -85,B 0,C 180,E1 -5236.625,E2 -5236.625} C_VEL
LIN {X 0,Y 519.364,Z 325.877,A -85,B 0,C 180,E1 -5237.422,E2 -5237.422} C_VEL
LIN {X 0,Y 519.799,Z 311.758,A -85,B 0,C 180,E1 -5238.118,E2 -5238.118} C_VEL
LIN {X 0,Y 520.156,Z 296.267,A -85,B 0,C 180,E1 -5238.704,E2 -5238.704} C_VEL
LIN {X 0,Y 520.434,Z 280.745,A -85,B 0,C 180,E1 -5239.115,E2 -5239.115} C_VEL
LIN {X 0,Y 520.635,Z 257.248,A -85,B 0,C 180,E1 -5239.492,E2 -5239.492} C_VEL
LIN {X 0,Y 521.925,Z 127.271,A -85,B 0,C 180,E1 -5241.442,E2 -5241.442} C_VEL
LIN {X 0,Y 519.175,Z 115.81,A -85,B 0,C 180,E1 -5241.741,E2 -5241.741} C_VEL
LIN {X 0,Y 518.27,Z 113.28,A -85,B 0,C 180,E1 -5241.821,E2 -5241.821} C_VEL
LIN {X 0,Y 516.899,Z 106.724,A -85,B 0,C 180,E1 -5242.912,E2 -5242.912} C_VEL
LIN {X 0,Y 516.895,Z 106.724,A -85,B 0,C 180,E1 -5246.185,E2 -5246.185} C_VEL
LIN {X 0,Y 516.871,Z 106.723,A -85,B 0,C 180,E1 -5248.966,E2 -5248.966} C_VEL
LIN {X 0,Y 516.233,Z 106.809,A -85,B 0,C 180,E1 -5249.617,E2 -5249.617} C_VEL
LIN {X 0,Y 513.355,Z 107.164,A -85,B 0,C 180,E1 -5250.673,E2 -5250.673} C_VEL
LIN {X 0,Y 510.923,Z 107.47,A -85,B 0,C 180,E1 -5251.524,E2 -5251.524} C_VEL
LIN {X 0,Y 509.912,Z 107.591,A -85,B 0,C 180,E1 -5252.181,E2 -5252.181} C_VEL
LIN {X 0,Y 509.849,Z 107.597,A -85,B 0,C 180,E1 -5252.404,E2 -5252.404} C_VEL
LIN {X 0,Y 509.823,Z 107.608,A -85,B 0,C 180,E1 -5255.578,E2 -5255.578} C_VEL
LIN {X 0,Y 509.85,Z 107.597,A -85,B 0,C 180,E1 -5258.339,E2 -5258.339} C_VEL
LIN {X 0,Y 509.81,Z 107.61,A -85,B 0,C 180,E1 -5261.431,E2 -5261.431} C_VEL
LIN {X 0,Y 509.841,Z 107.596,A -85,B 0,C 180,E1 -5264.67,E2 -5264.67} C_VEL
LIN {X 0,Y 509.793,Z 107.604,A -85,B 0,C 180,E1 -5267.506,E2 -5267.506} C_VEL
LIN {X 0,Y 509.834,Z 107.601,A -85,B 0,C 180,E1 -5270.646,E2 -5270.646} C_VEL
LIN {X 0,Y 509.811,Z 107.595,A -85,B 0,C 180,E1 -5273.646,E2 -5273.646} C_VEL
LIN {X 0,Y 509.841,Z 107.598,A -85,B 0,C 180,E1 -5276.538,E2 -5276.538} C_VEL
LIN {X 0,Y 509.822,Z 107.599,A -85,B 0,C 180,E1 -5279.333,E2 -5279.333} C_VEL
LIN {X 0,Y 509.833,Z 107.597,A -85,B 0,C 180,E1 -5282.051,E2 -5282.051} C_VEL
LIN {X 0,Y 509.804,Z 107.608,A -85,B 0,C 180,E1 -5284.7,E2 -5284.7} C_VEL
LIN {X 0,Y 509.827,Z 107.6,A -85,B 0,C 180,E1 -5287.459,E2 -5287.459} C_VEL
LIN {X 0,Y 509.893,Z 107.589,A -85,B 0,C 180,E1 -5289.844,E2 -5289.844} C_VEL
LIN {X 0,Y 509.855,Z 107.601,A -85,B 0,C 180,E1 -5292.347,E2 -5292.347} C_VEL
LIN {X 0,Y 509.888,Z 107.598,A -85,B 0,C 180,E1 -5294.818,E2 -5294.818} C_VEL
LIN {X 0,Y 509.905,Z 107.594,A -85,B 0,C 180,E1 -5298.124,E2 -5298.124} C_VEL
LIN {X 0,Y 509.877,Z 107.594,A -85,B 0,C 180,E1 -5301.279,E2 -5301.279} C_VEL
LIN {X 0,Y 509.9,Z 107.593,A -85,B 0,C 180,E1 -5303.669,E2 -5303.669} C_VEL
LIN {X 0,Y 509.887,Z 107.597,A -85,B 0,C 180,E1 -5306.839,E2 -5306.839} C_VEL
LIN {X 0,Y 509.926,Z 107.595,A -85,B 0,C 180,E1 -5308.42,E2 -5308.42} C_VEL
LIN {X 0,Y 509.949,Z 107.732,A -85,B 0,C 180,E1 -5310.271,E2 -5310.271} C_VEL
LIN {X 0,Y 512.617,Z 120.581,A -85,B 0,C 180,E1 -5312.161,E2 -5312.161} C_VEL
LIN {X 0,Y 512.151,Z 141.076,A -85,B 0,C 180,E1 -5314.933,E2 -5314.933} C_VEL
LIN {X 0,Y 512.295,Z 142.33,A -85,B 0,C 180,E1 -5315.001,E2 -5315.001} C_VEL
LIN {X 0,Y 515.279,Z 155.779,A -85,B 0,C 180,E1 -5315.334,E2 -5315.334} C_VEL
LIN {X 0,Y 514.096,Z 307.678,A -85,B 0,C 180,E1 -5317.536,E2 -5317.536} C_VEL
LIN {X 0,Y 513.814,Z 322.745,A -85,B 0,C 180,E1 -5317.911,E2 -5317.911} C_VEL
LIN {X 0,Y 513.454,Z 336.877,A -85,B 0,C 180,E1 -5318.412,E2 -5318.412} C_VEL
LIN {X 0,Y 512.999,Z 349.99,A -85,B 0,C 180,E1 -5319.015,E2 -5319.015} C_VEL
LIN {X 0,Y 512.433,Z 364.638,A -85,B 0,C 180,E1 -5319.871,E2 -5319.871} C_VEL
LIN {X 0,Y 511.929,Z 377.25,A -85,B 0,C 180,E1 -5320.781,E2 -5320.781} C_VEL
LIN {X 0,Y 511.324,Z 390.05,A -85,B 0,C 180,E1 -5321.898,E2 -5321.898} C_VEL
LIN {X 0,Y 510.809,Z 401.666,A -85,B 0,C 180,E1 -5323.121,E2 -5323.121} C_VEL
LIN {X 0,Y 510.333,Z 411.535,A -85,B 0,C 180,E1 -5324.352,E2 -5324.352} C_VEL
LIN {X 0,Y 509.957,Z 421.208,A -85,B 0,C 180,E1 -5325.8,E2 -5325.8} C_VEL
LIN {X 0,Y 509.669,Z 429.192,A -85,B 0,C 180,E1 -5327.246,E2 -5327.246} C_VEL
LIN {X 0,Y 509.505,Z 434.989,A -85,B 0,C 180,E1 -5328.497,E2 -5328.497} C_VEL
LIN {X 0,Y 509.373,Z 439.827,A -85,B 0,C 180,E1 -5329.757,E2 -5329.757} C_VEL
LIN {X 0,Y 509.261,Z 445.017,A -85,B 0,C 180,E1 -5331.451,E2 -5331.451} C_VEL
LIN {X 0,Y 509.155,Z 447.977,A -85,B 0,C 180,E1 -5332.736,E2 -5332.736} C_VEL
LIN {X 0,Y 509.078,Z 450.727,A -85,B 0,C 180,E1 -5334.467,E2 -5334.467} C_VEL
LIN {X 0,Y 509.073,Z 452.043,A -85,B 0,C 180,E1 -5336.217,E2 -5336.217} C_VEL
LIN {X 0,Y 509.086,Z 452.03,A -85,B 0,C 180,E1 -5337.928,E2 -5337.928} C_VEL
LIN {X 0,Y 509.116,Z 450.506,A -85,B 0,C 180,E1 -5339.799,E2 -5339.799} C_VEL
LIN {X 0,Y 509.154,Z 448.403,A -85,B 0,C 180,E1 -5341.151,E2 -5341.151} C_VEL
LIN {X 0,Y 509.219,Z 444.993,A -85,B 0,C 180,E1 -5342.659,E2 -5342.659} C_VEL
LIN {X 0,Y 509.347,Z 440.602,A -85,B 0,C 180,E1 -5344.117,E2 -5344.117} C_VEL
LIN {X 0,Y 509.478,Z 435.315,A -85,B 0,C 180,E1 -5345.523,E2 -5345.523} C_VEL
LIN {X 0,Y 509.712,Z 428.026,A -85,B 0,C 180,E1 -5347.086,E2 -5347.086} C_VEL
LIN {X 0,Y 510.02,Z 419.48,A -85,B 0,C 180,E1 -5348.575,E2 -5348.575} C_VEL
LIN {X 0,Y 510.375,Z 410.496,A -85,B 0,C 180,E1 -5349.886,E2 -5349.886} C_VEL
LIN {X 0,Y 510.887,Z 399.967,A -85,B 0,C 180,E1 -5351.173,E2 -5351.173} C_VEL
LIN {X 0,Y 511.384,Z 388.677,A -85,B 0,C 180,E1 -5352.331,E2 -5352.331} C_VEL
LIN {X 0,Y 511.91,Z 376.833,A -85,B 0,C 180,E1 -5353.35,E2 -5353.35} C_VEL
LIN {X 0,Y 512.495,Z 363.32,A -85,B 0,C 180,E1 -5354.309,E2 -5354.309} C_VEL
LIN {X 0,Y 513.035,Z 349.579,A -85,B 0,C 180,E1 -5355.098,E2 -5355.098} C_VEL
LIN {X 0,Y 513.482,Z 335.7,A -85,B 0,C 180,E1 -5355.73,E2 -5355.73} C_VEL
LIN {X 0,Y 513.855,Z 320.509,A -85,B 0,C 180,E1 -5356.247,E2 -5356.247} C_VEL
LIN {X 0,Y 514.108,Z 305.803,A -85,B 0,C 180,E1 -5356.591,E2 -5356.591} C_VEL
LIN {X 0,Y 515.271,Z 152.55,A -85,B 0,C 180,E1 -5358.805,E2 -5358.805} C_VEL
LIN {X 0,Y 513.005,Z 139.826,A -85,B 0,C 180,E1 -5359.111,E2 -5359.111} C_VEL
LIN {X 0,Y 513.41,Z 122.141,A -85,B 0,C 180,E1 -5360.973,E2 -5360.973} C_VEL
LIN {X 0,Y 509.85,Z 107.603,A -85,B 0,C 180,E1 -5362.696,E2 -5362.696} C_VEL
LIN {X 0,Y 509.858,Z 107.602,A -85,B 0,C 180,E1 -5365.797,E2 -5365.797} C_VEL
LIN {X 0,Y 509.848,Z 107.599,A -85,B 0,C 180,E1 -5368.72,E2 -5368.72} C_VEL
LIN {X 0,Y 509.899,Z 107.597,A -85,B 0,C 180,E1 -5371.899,E2 -5371.899} C_VEL
LIN {X 0,Y 509.879,Z 107.597,A -85,B 0,C 180,E1 -5374.704,E2 -5374.704} C_VEL
LIN {X 0,Y 509.858,Z 107.712,A -85,B 0,C 180,E1 -5377.243,E2 -5377.243} C_VEL
LIN {X 0,Y 511.081,Z 112.739,A -85,B 0,C 180,E1 -5377.929,E2 -5377.929} C_VEL
LIN {X 0,Y 515.027,Z 123.402,A -85,B 0,C 180,E1 -5378.28,E2 -5378.28} C_VEL
LIN {X 0,Y 515.311,Z 126.362,A -85,B 0,C 180,E1 -5378.341,E2 -5378.341} C_VEL
LIN {X 0,Y 513.693,Z 279.491,A -85,B 0,C 180,E1 -5380.702,E2 -5380.702} C_VEL
LIN {X 0,Y 513.444,Z 294.911,A -85,B 0,C 180,E1 -5381.101,E2 -5381.101} C_VEL
LIN {X 0,Y 513.07,Z 309.541,A -85,B 0,C 180,E1 -5381.636,E2 -5381.636} C_VEL
LIN {X 0,Y 512.678,Z 322.273,A -85,B 0,C 180,E1 -5382.241,E2 -5382.241} C_VEL
LIN {X 0,Y 512.183,Z 335.961,A -85,B 0,C 180,E1 -5383.047,E2 -5383.047} C_VEL
LIN {X 0,Y 511.647,Z 349.843,A -85,B 0,C 180,E1 -5384.054,E2 -5384.054} C_VEL
LIN {X 0,Y 511.182,Z 362.356,A -85,B 0,C 180,E1 -5385.163,E2 -5385.163} C_VEL
LIN {X 0,Y 510.747,Z 372.81,A -85,B 0,C 180,E1 -5386.269,E2 -5386.269} C_VEL
LIN {X 0,Y 510.331,Z 382.494,A -85,B 0,C 180,E1 -5387.473,E2 -5387.473} C_VEL
LIN {X 0,Y 510.021,Z 391.965,A -85,B 0,C 180,E1 -5388.877,E2 -5388.877} C_VEL
LIN {X 0,Y 509.716,Z 399.827,A -85,B 0,C 180,E1 -5390.276,E2 -5390.276} C_VEL
LIN {X 0,Y 509.536,Z 406.339,A -85,B 0,C 180,E1 -5391.673,E2 -5391.673} C_VEL
LIN {X 0,Y 509.415,Z 410.934,A -85,B 0,C 180,E1 -5392.867,E2 -5392.867} C_VEL
LIN {X 0,Y 509.325,Z 415.826,A -85,B 0,C 180,E1 -5394.457,E2 -5394.457} C_VEL
LIN {X 0,Y 509.258,Z 419.419,A -85,B 0,C 180,E1 -5396.043,E2 -5396.043} C_VEL
LIN {X 0,Y 509.196,Z 421.802,A -85,B 0,C 180,E1 -5397.627,E2 -5397.627} C_VEL
LIN {X 0,Y 509.089,Z 423.035,A -85,B 0,C 180,E1 -5399.209,E2 -5399.209} C_VEL
LIN {X 0,Y 509.091,Z 423.089,A -85,B 0,C 180,E1 -5400.791,E2 -5400.791} C_VEL
LIN {X 0,Y 509.196,Z 421.979,A -85,B 0,C 180,E1 -5402.373,E2 -5402.373} C_VEL
LIN {X 0,Y 509.262,Z 419.717,A -85,B 0,C 180,E1 -5403.956,E2 -5403.956} C_VEL
LIN {X 0,Y 509.33,Z 416.243,A -85,B 0,C 180,E1 -5405.543,E2 -5405.543} C_VEL
LIN {X 0,Y 509.441,Z 411.469,A -85,B 0,C 180,E1 -5407.132,E2 -5407.132} C_VEL
LIN {X 0,Y 509.587,Z 405.261,A -85,B 0,C 180,E1 -5408.726,E2 -5408.726} C_VEL
LIN {X 0,Y 509.825,Z 397.413,A -85,B 0,C 180,E1 -5410.323,E2 -5410.323} C_VEL
LIN {X 0,Y 510.1,Z 389.059,A -85,B 0,C 180,E1 -5411.716,E2 -5411.716} C_VEL
LIN {X 0,Y 510.465,Z 380.417,A -85,B 0,C 180,E1 -5412.928,E2 -5412.928} C_VEL
LIN {X 0,Y 510.881,Z 370.209,A -85,B 0,C 180,E1 -5414.133,E2 -5414.133} C_VEL
LIN {X 0,Y 511.344,Z 358.31,A -85,B 0,C 180,E1 -5415.313,E2 -5415.313} C_VEL
LIN {X 0,Y 511.808,Z 345.709,A -85,B 0,C 180,E1 -5416.349,E2 -5416.349} C_VEL
LIN {X 0,Y 512.274,Z 332.256,A -85,B 0,C 180,E1 -5417.258,E2 -5417.258} C_VEL
LIN {X 0,Y 512.716,Z 317.319,A -85,B 0,C 180,E1 -5418.067,E2 -5418.067} C_VEL
LIN {X 0,Y 513.146,Z 302,A -85,B 0,C 180,E1 -5418.699,E2 -5418.699} C_VEL
LIN {X 0,Y 513.405,Z 286.95,A -85,B 0,C 180,E1 -5419.154,E2 -5419.154} C_VEL
LIN {X 0,Y 513.562,Z 271.547,A -85,B 0,C 180,E1 -5419.459,E2 -5419.459} C_VEL
LIN {X 0,Y 514.886,Z 165.788,A -85,B 0,C 180,E1 -5421.128,E2 -5421.128} C_VEL
LIN {X 0,Y 515.277,Z 127.384,A -85,B 0,C 180,E1 -5421.779,E2 -5421.779} C_VEL
LIN {X 0,Y 512.906,Z 119.217,A -85,B 0,C 180,E1 -5422.046,E2 -5422.046} C_VEL
LIN {X 0,Y 511.98,Z 117.004,A -85,B 0,C 180,E1 -5422.14,E2 -5422.14} C_VEL
LIN {X 0,Y 509.837,Z 107.606,A -85,B 0,C 180,E1 -5424.048,E2 -5424.048} C_VEL
LIN {X 0,Y 509.846,Z 107.603,A -85,B 0,C 180,E1 -5427.058,E2 -5427.058} C_VEL
LIN {X 0,Y 509.851,Z 107.604,A -85,B 0,C 180,E1 -5429.751,E2 -5429.751} C_VEL
LIN {X 0,Y 509.845,Z 107.601,A -85,B 0,C 180,E1 -5432.769,E2 -5432.769} C_VEL
LIN {X 0,Y 509.82,Z 107.608,A -85,B 0,C 180,E1 -5435.577,E2 -5435.577} C_VEL
LIN {X 0,Y 509.848,Z 107.599,A -85,B 0,C 180,E1 -5438.338,E2 -5438.338} C_VEL
LIN {X 0,Y 509.806,Z 107.609,A -85,B 0,C 180,E1 -5441.43,E2 -5441.43} C_VEL
LIN {X 0,Y 509.838,Z 107.602,A -85,B 0,C 180,E1 -5444.67,E2 -5444.67} C_VEL
LIN {X 0,Y 509.79,Z 107.61,A -85,B 0,C 180,E1 -5447.506,E2 -5447.506} C_VEL
LIN {X 0,Y 509.831,Z 107.604,A -85,B 0,C 180,E1 -5450.646,E2 -5450.646} C_VEL
LIN {X 0,Y 509.801,Z 107.608,A -85,B 0,C 180,E1 -5453.645,E2 -5453.645} C_VEL
LIN {X 0,Y 509.837,Z 107.606,A -85,B 0,C 180,E1 -5456.537,E2 -5456.537} C_VEL
LIN {X 0,Y 509.813,Z 107.61,A -85,B 0,C 180,E1 -5459.79,E2 -5459.79} C_VEL
LIN {X 0,Y 509.813,Z 107.735,A -85,B 0,C 180,E1 -5460.189,E2 -5460.189} C_VEL
LIN {X 0,Y 513.093,Z 121.025,A -85,B 0,C 180,E1 -5462.244,E2 -5462.244} C_VEL
LIN {X 0,Y 513.204,Z 125.807,A -85,B 0,C 180,E1 -5462.89,E2 -5462.89} C_VEL
LIN {X 0,Y 512.404,Z 145.941,A -85,B 0,C 180,E1 -5465.487,E2 -5465.487} C_VEL
LIN {X 0,Y 511.82,Z 164.898,A -85,B 0,C 180,E1 -5467.859,E2 -5467.859} C_VEL
LIN {X 0,Y 515.098,Z 184.586,A -85,B 0,C 180,E1 -5468.355,E2 -5468.355} C_VEL
LIN {X 0,Y 513.762,Z 292.988,A -85,B 0,C 180,E1 -5470.08,E2 -5470.08} C_VEL
LIN {X 0,Y 513.354,Z 333.545,A -85,B 0,C 180,E1 -5470.714,E2 -5470.714} C_VEL
LIN {X 0,Y 512.968,Z 349.441,A -85,B 0,C 180,E1 -5471.119,E2 -5471.119} C_VEL
LIN {X 0,Y 512.595,Z 364.608,A -85,B 0,C 180,E1 -5471.67,E2 -5471.67} C_VEL
LIN {X 0,Y 512.114,Z 378.507,A -85,B 0,C 180,E1 -5472.324,E2 -5472.324} C_VEL
LIN {X 0,Y 511.632,Z 392.199,A -85,B 0,C 180,E1 -5473.131,E2 -5473.131} C_VEL
LIN {X 0,Y 511.147,Z 406.352,A -85,B 0,C 180,E1 -5474.161,E2 -5474.161} C_VEL
LIN {X 0,Y 510.697,Z 418.745,A -85,B 0,C 180,E1 -5475.251,E2 -5475.251} C_VEL
LIN {X 0,Y 510.278,Z 430.25,A -85,B 0,C 180,E1 -5476.459,E2 -5476.459} C_VEL
LIN {X 0,Y 509.973,Z 439.931,A -85,B 0,C 180,E1 -5477.666,E2 -5477.666} C_VEL
LIN {X 0,Y 509.696,Z 449.407,A -85,B 0,C 180,E1 -5479.071,E2 -5479.071} C_VEL
LIN {X 0,Y 509.462,Z 457.248,A -85,B 0,C 180,E1 -5480.471,E2 -5480.471} C_VEL
LIN {X 0,Y 509.354,Z 464.559,A -85,B 0,C 180,E1 -5482.069,E2 -5482.069} C_VEL
LIN {X 0,Y 509.285,Z 470.294,A -85,B 0,C 180,E1 -5483.662,E2 -5483.662} C_VEL
LIN {X 0,Y 509.159,Z 474.618,A -85,B 0,C 180,E1 -5485.249,E2 -5485.249} C_VEL
LIN {X 0,Y 509.189,Z 477.661,A -85,B 0,C 180,E1 -5486.835,E2 -5486.835} C_VEL
LIN {X 0,Y 509.11,Z 479.48,A -85,B 0,C 180,E1 -5488.418,E2 -5488.418} C_VEL
LIN {X 0,Y 509.077,Z 480.116,A -85,B 0,C 180,E1 -5490,E2 -5490} C_VEL
LIN {X 0,Y 509.11,Z 479.523,A -85,B 0,C 180,E1 -5491.582,E2 -5491.582} C_VEL
LIN {X 0,Y 509.189,Z 477.753,A -85,B 0,C 180,E1 -5493.165,E2 -5493.165} C_VEL
LIN {X 0,Y 509.159,Z 474.77,A -85,B 0,C 180,E1 -5494.751,E2 -5494.751} C_VEL
LIN {X 0,Y 509.285,Z 470.515,A -85,B 0,C 180,E1 -5496.338,E2 -5496.338} C_VEL
LIN {X 0,Y 509.356,Z 464.859,A -85,B 0,C 180,E1 -5497.931,E2 -5497.931} C_VEL
LIN {X 0,Y 509.463,Z 457.654,A -85,B 0,C 180,E1 -5499.529,E2 -5499.529} C_VEL
LIN {X 0,Y 509.699,Z 449.938,A -85,B 0,C 180,E1 -5500.929,E2 -5500.929} C_VEL
LIN {X 0,Y 509.983,Z 440.637,A -85,B 0,C 180,E1 -5502.334,E2 -5502.334} C_VEL
LIN {X 0,Y 510.329,Z 431.132,A -85,B 0,C 180,E1 -5503.54,E2 -5503.54} C_VEL
LIN {X 0,Y 510.827,Z 418.881,A -85,B 0,C 180,E1 -5504.847,E2 -5504.847} C_VEL
LIN {X 0,Y 511.283,Z 406.357,A -85,B 0,C 180,E1 -5505.957,E2 -5505.957} C_VEL
LIN {X 0,Y 511.747,Z 394.029,A -85,B 0,C 180,E1 -5506.865,E2 -5506.865} C_VEL
LIN {X 0,Y 512.268,Z 380.784,A -85,B 0,C 180,E1 -5507.67,E2 -5507.67} C_VEL
LIN {X 0,Y 512.778,Z 366.363,A -85,B 0,C 180,E1 -5508.375,E2 -5508.375} C_VEL
LIN {X 0,Y 513.208,Z 351.242,A -85,B 0,C 180,E1 -5508.939,E2 -5508.939} C_VEL
LIN {X 0,Y 513.561,Z 336.504,A -85,B 0,C 180,E1 -5509.33,E2 -5509.33} C_VEL
LIN {X 0,Y 513.839,Z 312.016,A -85,B 0,C 180,E1 -5509.734,E2 -5509.734} C_VEL
LIN {X 0,Y 515.107,Z 189.197,A -85,B 0,C 180,E1 -5511.596,E2 -5511.596} C_VEL
LIN {X 0,Y 514.93,Z 179.454,A -85,B 0,C 180,E1 -5511.762,E2 -5511.762} C_VEL
LIN {X 0,Y 512.821,Z 165.334,A -85,B 0,C 180,E1 -5512.098,E2 -5512.098} C_VEL
LIN {X 0,Y 513.637,Z 140.3,A -85,B 0,C 180,E1 -5514.558,E2 -5514.558} C_VEL
LIN {X 0,Y 514.297,Z 124.241,A -85,B 0,C 180,E1 -5516.149,E2 -5516.149} C_VEL
LIN {X 0,Y 509.82,Z 107.606,A -85,B 0,C 180,E1 -5518.121,E2 -5518.121} C_VEL
LIN {X 0,Y 509.827,Z 107.606,A -85,B 0,C 180,E1 -5520.667,E2 -5520.667} C_VEL
LIN {X 0,Y 509.837,Z 107.602,A -85,B 0,C 180,E1 -5523.463,E2 -5523.463} C_VEL
LIN {X 0,Y 509.807,Z 107.605,A -85,B 0,C 180,E1 -5526.355,E2 -5526.355} C_VEL
LIN {X 0,Y 509.831,Z 107.603,A -85,B 0,C 180,E1 -5529.354,E2 -5529.354} C_VEL
LIN {X 0,Y 509.79,Z 107.608,A -85,B 0,C 180,E1 -5532.494,E2 -5532.494} C_VEL
LIN {X 0,Y 509.838,Z 107.598,A -85,B 0,C 180,E1 -5535.33,E2 -5535.33} C_VEL
LIN {X 0,Y 509.806,Z 107.609,A -85,B 0,C 180,E1 -5538.57,E2 -5538.57} C_VEL
LIN {X 0,Y 509.848,Z 107.599,A -85,B 0,C 180,E1 -5541.787,E2 -5541.787} C_VEL
LIN {X 0,Y 509.824,Z 107.608,A -85,B 0,C 180,E1 -5544.622,E2 -5544.622} C_VEL
LIN {X 0,Y 509.859,Z 107.598,A -85,B 0,C 180,E1 -5547.481,E2 -5547.481} C_VEL
LIN {X 0,Y 509.853,Z 107.604,A -85,B 0,C 180,E1 -5550.275,E2 -5550.275} C_VEL
LIN {X 0,Y 509.825,Z 107.605,A -85,B 0,C 180,E1 -5552.941,E2 -5552.941} C_VEL
LIN {X 0,Y 509.835,Z 107.605,A -85,B 0,C 180,E1 -5555.572,E2 -5555.572} C_VEL
LIN {X 0,Y 509.835,Z 107.695,A -85,B 0,C 180,E1 -5556.706,E2 -5556.706} C_VEL
LIN {X 0,Y 511.755,Z 115.747,A -85,B 0,C 180,E1 -5557.947,E2 -5557.947} C_VEL
LIN {X 0,Y 514.099,Z 122.6,A -85,B 0,C 180,E1 -5558.191,E2 -5558.191} C_VEL
LIN {X 0,Y 515.321,Z 127.987,A -85,B 0,C 180,E1 -5558.347,E2 -5558.347} C_VEL
LIN {X 0,Y 513.967,Z 230.361,A -85,B 0,C 180,E1 -5560.011,E2 -5560.011} C_VEL
LIN {X 0,Y 513.487,Z 280.524,A -85,B 0,C 180,E1 -5560.803,E2 -5560.803} C_VEL
LIN {X 0,Y 513.22,Z 296.077,A -85,B 0,C 180,E1 -5561.203,E2 -5561.203} C_VEL
LIN {X 0,Y 512.879,Z 310.512,A -85,B 0,C 180,E1 -5561.733,E2 -5561.733} C_VEL
LIN {X 0,Y 512.567,Z 323.287,A -85,B 0,C 180,E1 -5562.34,E2 -5562.34} C_VEL
LIN {X 0,Y 512.092,Z 336.994,A -85,B 0,C 180,E1 -5563.147,E2 -5563.147} C_VEL
LIN {X 0,Y 511.646,Z 349.583,A -85,B 0,C 180,E1 -5564.055,E2 -5564.055} C_VEL
LIN {X 0,Y 511.159,Z 362.274,A -85,B 0,C 180,E1 -5565.163,E2 -5565.163} C_VEL
LIN {X 0,Y 510.768,Z 372.866,A -85,B 0,C 180,E1 -5566.27,E2 -5566.27} C_VEL
LIN {X 0,Y 510.379,Z 382.78,A -85,B 0,C 180,E1 -5567.495,E2 -5567.495} C_VEL
LIN {X 0,Y 510.043,Z 392.139,A -85,B 0,C 180,E1 -5568.878,E2 -5568.878} C_VEL
LIN {X 0,Y 509.753,Z 399.008,A -85,B 0,C 180,E1 -5570.076,E2 -5570.076} C_VEL
LIN {X 0,Y 509.568,Z 406.525,A -85,B 0,C 180,E1 -5571.674,E2 -5571.674} C_VEL
LIN {X 0,Y 509.441,Z 411.073,A -85,B 0,C 180,E1 -5572.868,E2 -5572.868} C_VEL
LIN {X 0,Y 509.329,Z 415.937,A -85,B 0,C 180,E1 -5574.457,E2 -5574.457} C_VEL
LIN {X 0,Y 509.258,Z 419.49,A -85,B 0,C 180,E1 -5576.044,E2 -5576.044} C_VEL
LIN {X 0,Y 509.196,Z 421.829,A -85,B 0,C 180,E1 -5577.627,E2 -5577.627} C_VEL
LIN {X 0,Y 509.087,Z 423.012,A -85,B 0,C 180,E1 -5579.209,E2 -5579.209} C_VEL
LIN {X 0,Y 509.087,Z 423.005,A -85,B 0,C 180,E1 -5580.791,E2 -5580.791} C_VEL
LIN {X 0,Y 509.196,Z 421.844,A -85,B 0,C 180,E1 -5582.373,E2 -5582.373} C_VEL
LIN {X 0,Y 509.258,Z 419.53,A -85,B 0,C 180,E1 -5583.957,E2 -5583.957} C_VEL
LIN {X 0,Y 509.324,Z 416.004,A -85,B 0,C 180,E1 -5585.543,E2 -5585.543} C_VEL
LIN {X 0,Y 509.408,Z 411.183,A -85,B 0,C 180,E1 -5587.133,E2 -5587.133} C_VEL
LIN {X 0,Y 509.565,Z 404.934,A -85,B 0,C 180,E1 -5588.727,E2 -5588.727} C_VEL
LIN {X 0,Y 509.784,Z 397.066,A -85,B 0,C 180,E1 -5590.325,E2 -5590.325} C_VEL
LIN {X 0,Y 510.058,Z 388.254,A -85,B 0,C 180,E1 -5591.786,E2 -5591.786} C_VEL
LIN {X 0,Y 510.515,Z 378.479,A -85,B 0,C 180,E1 -5593.129,E2 -5593.129} C_VEL
LIN {X 0,Y 510.937,Z 368.048,A -85,B 0,C 180,E1 -5594.335,E2 -5594.335} C_VEL
LIN {X 0,Y 511.406,Z 356.32,A -85,B 0,C 180,E1 -5595.474,E2 -5595.474} C_VEL
LIN {X 0,Y 511.87,Z 344.322,A -85,B 0,C 180,E1 -5596.451,E2 -5596.451} C_VEL
LIN {X 0,Y 512.37,Z 330.808,A -85,B 0,C 180,E1 -5597.358,E2 -5597.358} C_VEL
LIN {X 0,Y 512.813,Z 316.824,A -85,B 0,C 180,E1 -5598.115,E2 -5598.115} C_VEL
LIN {X 0,Y 513.257,Z 301.812,A -85,B 0,C 180,E1 -5598.746,E2 -5598.746} C_VEL
LIN {X 0,Y 513.544,Z 287.185,A -85,B 0,C 180,E1 -5599.201,E2 -5599.201} C_VEL
LIN {X 0,Y 513.746,Z 271.247,A -85,B 0,C 180,E1 -5599.53,E2 -5599.53} C_VEL
LIN {X 0,Y 515.21,Z 133.749,A -85,B 0,C 180,E1 -5601.626,E2 -5601.626} C_VEL
LIN {X 0,Y 515.12,Z 127.555,A -85,B 0,C 180,E1 -5601.73,E2 -5601.73} C_VEL
LIN {X 0,Y 512.776,Z 118.095,A -85,B 0,C 180,E1 -5601.986,E2 -5601.986} C_VEL
LIN {X 0,Y 511.119,Z 113.433,A -85,B 0,C 180,E1 -5602.147,E2 -5602.147} C_VEL
LIN {X 0,Y 509.849,Z 107.603,A -85,B 0,C 180,E1 -5603.132,E2 -5603.132} C_VEL
LIN {X 0,Y 509.853,Z 107.599,A -85,B 0,C 180,E1 -5606.365,E2 -5606.365} C_VEL
LIN {X 0,Y 509.835,Z 107.599,A -85,B 0,C 180,E1 -5608.963,E2 -5608.963} C_VEL
LIN {X 0,Y 509.82,Z 107.608,A -85,B 0,C 180,E1 -5611.591,E2 -5611.591} C_VEL
LIN {X 0,Y 509.849,Z 107.597,A -85,B 0,C 180,E1 -5612.404,E2 -5612.404} C_VEL
LIN {X 0,Y 509.229,Z 107.677,A -85,B 0,C 180,E1 -5613.063,E2 -5613.063} C_VEL
LIN {X 0,Y 506.372,Z 108.038,A -85,B 0,C 180,E1 -5614.133,E2 -5614.133} C_VEL
LIN {X 0,Y 503.92,Z 108.345,A -85,B 0,C 180,E1 -5614.996,E2 -5614.996} C_VEL
LIN {X 0,Y 502.859,Z 108.475,A -85,B 0,C 180,E1 -5615.662,E2 -5615.662} C_VEL
LIN {X 0,Y 502.77,Z 108.483,A -85,B 0,C 180,E1 -5615.888,E2 -5615.888} C_VEL
LIN {X 0,Y 502.795,Z 108.478,A -85,B 0,C 180,E1 -5618.977,E2 -5618.977} C_VEL
LIN {X 0,Y 502.773,Z 108.478,A -85,B 0,C 180,E1 -5622.195,E2 -5622.195} C_VEL
LIN {X 0,Y 502.787,Z 108.472,A -85,B 0,C 180,E1 -5625.47,E2 -5625.47} C_VEL
LIN {X 0,Y 502.766,Z 108.479,A -85,B 0,C 180,E1 -5628.929,E2 -5628.929} C_VEL
LIN {X 0,Y 502.792,Z 108.475,A -85,B 0,C 180,E1 -5632.046,E2 -5632.046} C_VEL
LIN {X 0,Y 502.794,Z 108.474,A -85,B 0,C 180,E1 -5635.034,E2 -5635.034} C_VEL
LIN {X 0,Y 502.78,Z 108.477,A -85,B 0,C 180,E1 -5637.915,E2 -5637.915} C_VEL
LIN {X 0,Y 502.793,Z 108.476,A -85,B 0,C 180,E1 -5640.71,E2 -5640.71} C_VEL
LIN {X 0,Y 502.777,Z 108.479,A -85,B 0,C 180,E1 -5643.46,E2 -5643.46} C_VEL
LIN {X 0,Y 502.763,Z 108.475,A -85,B 0,C 180,E1 -5646.085,E2 -5646.085} C_VEL
LIN {X 0,Y 502.833,Z 108.469,A -85,B 0,C 180,E1 -5649.464,E2 -5649.464} C_VEL
LIN {X 0,Y 502.789,Z 108.479,A -85,B 0,C 180,E1 -5652.09,E2 -5652.09} C_VEL
LIN {X 0,Y 502.825,Z 108.473,A -85,B 0,C 180,E1 -5655.429,E2 -5655.429} C_VEL
LIN {X 0,Y 502.879,Z 108.469,A -85,B 0,C 180,E1 -5658.717,E2 -5658.717} C_VEL
LIN {X 0,Y 502.85,Z 108.473,A -85,B 0,C 180,E1 -5661.966,E2 -5661.966} C_VEL
LIN {X 0,Y 502.89,Z 108.473,A -85,B 0,C 180,E1 -5664.386,E2 -5664.386} C_VEL
LIN {X 0,Y 503.011,Z 108.454,A -85,B 0,C 180,E1 -5667.598,E2 -5667.598} C_VEL
LIN {X 0,Y 503.017,Z 108.586,A -85,B 0,C 180,E1 -5670.025,E2 -5670.025} C_VEL
LIN {X 0,Y 505.749,Z 121.893,A -85,B 0,C 180,E1 -5671.991,E2 -5671.991} C_VEL
LIN {X 0,Y 505.351,Z 141.308,A -85,B 0,C 180,E1 -5674.637,E2 -5674.637} C_VEL
LIN {X 0,Y 506.037,Z 144.913,A -85,B 0,C 180,E1 -5674.755,E2 -5674.755} C_VEL
LIN {X 0,Y 508.718,Z 157.797,A -85,B 0,C 180,E1 -5675.072,E2 -5675.072} C_VEL
LIN {X 0,Y 507.44,Z 307.172,A -85,B 0,C 180,E1 -5677.26,E2 -5677.26} C_VEL
LIN {X 0,Y 507.137,Z 321.724,A -85,B 0,C 180,E1 -5677.615,E2 -5677.615} C_VEL
LIN {X 0,Y 506.697,Z 337.361,A -85,B 0,C 180,E1 -5678.173,E2 -5678.173} C_VEL
